(* CODESYS project DEMO.export

Project tree, tasks and I/O mapping:
  Device : Haitian E112C-0808N, Ningbo Anson CNC Technique CO., Ltd., version 1.1.32.0
      unmapped channels: DI, IN0_1_COUNT, IN2_3_COUNT, IN4_5_COUNT, IN6_7_COUNT, DO, OUT0_1_Pluse, OUT2_3_Pluse, OUT4_5_Pluse, OUT6_7_Pluse, IN, OUT
    application Application
      libraries: Standard, 3.5.18.0 (System); E112C Motion Control Lib, * (Haitian); E112C Communication  Lib, * (Haitian)
      task EtherCAT_Task (cyclic, interval 1000 µs, priority 1) calls DriverInHandlersEthercat, DriverOutHandlersEthercat, InitAxesProgram
      task MainTask (cyclic, interval 1 ms, priority 1) calls Motion_IO, Motion, Punch_PA, prTestFunction, DebugMode
      task Task1 (cyclic, interval 10 ms, priority 2) calls ModbusTCP_MasterPRG, prHMI, prCoolFan, prHMI_Error, SDO_test, prIOsetting_test, prModusTcp_Fanuc, SetPosition
      data type AxAbs
      data type Def_1
      data type Tcp_1
      BAK/
        program Punch_PA_1 [ST]
      FunctionBlock/
        function block FB_BLINK [ST]
        function block FB_CrankSliderHeight [ST]
        function block FB_HeightToAngle [ST]
        function block FB_Toggle [ST]
      MosbusTcp/
        program Modbus_Client_Fanuc [LD]: ACT_TRIG
        program prHMI [ST]
        program prHMI_Error [ST]
        program prModusTcp_Fanuc [ST]
      global variables AxisVars
      global variables GVL_Axis
      global variables GVL_HMI
      global variables GVL_PA
      global variables ModbusTCP_MasterVars
      program DebugMode [ST]: act_MoveNegative, act_MovePositive, act_SetHome
      program DriverInHandlersEthercat [ST]
      program DriverOutHandlersEthercat [ST]
      program InitAxesProgram [ST]
      program ModbusTCP_MasterPRG [ST]
      program Motion [ST]
      program Motion_IO [ST]
      program prCoolFan [ST]
      program prIOsetting_test [LD]: act_EtherCAT_monitor, act_Tcpdata
      program prTestFunction [ST]: act_Jump_To_PTE
      program Punch_PA [ST]: act_20_PunchA_GoPOP, act_21_PunchA_PunchA, act_22_PunchA_PunchB, act_31_PunchAB_PunchA, act_33_PunchAB_PunchB, act_41_PunchSoft_PunchA1, act_42_PunchSoft_PunchA2, act_43_PunchSoft_PunchA3, act_45_PunchSoft_PunchB1, act_46_PunchSoft_PunchB2, act_47_PunchSoft_PunchB3, act_7_GoPTE, act_Jump_To_PTE
      program SDO_test [LD]: act_Blink
      program SetHome [FBD]
      program SetPosition [?]
      program SetPosition0 [LD]
      program Test_Crank [ST]
      trace Trace (task MainTask): AxisVars.Axis0.AxisMotionState.ActPosition, ibPunch, qbReadyFeed, DriverOutHandlersEthercat.DriveOutHandler_Axis0.SetPosition
      global variables PersistentVars
    设备诊断
    设备组态
      EtherCAT机架
    轴配置
    资源使用表
    HT_LocalIO
        unmapped channels: DI, IN0_1_COUNT, IN2_3_COUNT, IN4_5_COUNT, IN6_7_COUNT, DO, OUT0_1_Pluse, OUT2_3_Pluse, OUT4_5_Pluse, OUT6_7_Pluse
    HT_LocalBus
        settings: EModuleCycle = 1000 us
      EM-DO16P [DO16 PNP] : EM-DO16P [DO16 PNP], Haitian, version 1.1.32.0
          unmapped channels: DO, DO
    HT_EtherCAT
      HT_Hi Drive v5.0 (TMS320F28377S, 16Bit Async, ET1100) : HT_Hi Drive v5.0 (TMS320F28377S, 16Bit Async, ET1100), HAITIAN DRIVE CO.,LTD, order no. Hi Drive v5.0, version Revision=16#00000001
          input  Application.DriverInHandlersEthercat.DriveInHandler_Axis0.StatusWord : UINT  // Status Word
          input  Application.DriverInHandlersEthercat.DriveInHandler_Axis0.ActPosition : DINT  // Position actual value
          input  Application.DriverInHandlersEthercat.DriveInHandler_Axis0.ActTorque : INT  // CI06 Current Iq actual value [A]
          input  Application.DriverInHandlersEthercat.DriveInHandler_Axis0.ActVelocity : DINT  // Velocity actual value [/10 r/min]
          input  Application.DriverInHandlersEthercat.DriveInHandler_Axis0.ModeOfDisplay : SINT  // Modes of operation display
          output Application.DriverOutHandlersEthercat.DriveOutHandler_Axis0.ControlWord : UINT  // Control Word
          output Application.DriverOutHandlersEthercat.DriveOutHandler_Axis0.SetTorque : INT  // Target torque [/10 %]
          output Application.DriverOutHandlersEthercat.DriveOutHandler_Axis0.SetPosition : DINT  // Target position
          output Application.DriverOutHandlersEthercat.DriveOutHandler_Axis0.SetVelocity : DINT  // Target velocity
          output Application.DriverOutHandlersEthercat.DriveOutHandler_Axis0.ModeOfOperation : SINT  // Modes of operation
          unmapped channels: RU09 Motor temperature [°C], Drive Error Code*, Max torque [/10 %], Elements
    HT_Ethernet
        settings: ip.ip = 192; ip.ip = 168; ip.ip = 1; ip.ip = 66; netmask.netmask = 255; netmask.netmask = 255; netmask.netmask = 255; netmask.netmask = 0; gateway.gateway = 192; gateway.gateway = 168; gateway.gateway = 1; gateway.gateway = 254; ModbusSlaveAddr = 0
    HT_EX1
    HT_EX2
    HT_Elink
        unmapped channels: IN, OUT
    HT_RS485_1
    HT_RS485_2
*)

// Device/Application/AxAbs
TYPE AxAbs :
STRUCT
	bExe :BOOL;
	Position :LREAL;
	Speed :LREAL;
	Acc :LREAL;
	Dcc :LREAL;
	Jerk :LREAL;
	Dir :MC_DIRECTION;
	BufferMode :MC_BUFFER_MODE;
	Done :BOOL;
	Busy :BOOL;
	Aborted :BOOL;
	Error :BOOL;
	ErrorID :WORD;
	Active :BOOL;
END_STRUCT
END_TYPE

// Device/Application/Def_1
TYPE Def_1 :
STRUCT
	
	Speed_Go_PTE :REAL :=100; //Go上死点PTE 速度
	Speed_Go_POP :REAL :=100; //上死点到预压POP 速度
 	
	
	Acc_Go_PTE : REAL :=3600;
	Acc_Go_POP : REAL :=3600;
	Acc_PunchA : REAL :=36000; //冲压A side
	Acc_PunchAB : REAL :=360000; //冲压AB side
	Acc_PunchSoft : REAL :=100000; //软冲 side
	
	CoolFan_Toff :INT :=10; //延时风扇关闭 sec 
	CoolFan_OnTemp :INT :=60; //自动打开温度
	
	PTE_Gap :REAL :=5; //到上死点0的到位窗口
	POP_Gap :REAL :=3; //到预压位角度的到位窗口 不是提前到位信号
	PUP_Gap :REAL :=2; //到下死点角度的到位窗口 不是提前到位信号	
	POP_ReadyWin_Punch :REAL :=10; //冲头冲压返回预压位置的提前到位窗口信号
	POP_ReadyWin_Mark :REAL :=5; //冲头冲压返回预压位置的提前到位窗口信号
	PunchSpeed_Max_Lim :REAL :=425; //冲头最高速度限制值
END_STRUCT
END_TYPE

// Device/Application/Tcp_1
TYPE Tcp_1 :
STRUCT
	bError :BOOL; 
	iRead_OK :INT; //读取数据正常计数器
	
	iPTE_mm :REAL :=32; //Data_1 换模位置 
	iPTE_deg :REAL; //Data_1 换模位置

	iPOP_mm :REAL;//Data_2 预压位置 上死点
	iPOP_deg :REAL;//Data_2 预压位置 上死点
	
	iPUP_mm :REAL; //Data_3 下压位置
	iPUP_deg :REAL;//Data_3 下压位置

	iReady_mm :REAL; //Data_4换模位置 ready 信号区域
	iReady_deg :REAL;//Data_4换模位置 ready 信号区域
	
	iDelayTime_ms : UINT;//Data_5  下压点延时

	iPunchSpeed_Trans :REAL; //Data_6 冲压速度	
	iPunchSpeed_Max :REAL; //Data_6 冲压速度
	iSoftPunch : INT;//Data_7 软冲模式
	
	iPSP1_mm :REAL ;//Data_8 软冲减速点1
	iPSP1_deg :REAL ;//Data_8 软冲减速点1
	
	iPunchSpeed :REAL; //Data_9 冲压穿板速度
	
	iFormMode :INT; //Data_10 压印模式 0-可调 1-机械点
	
	iPSP2_mm :REAL ;//Data_11 软冲减速点1
	iPSP2_deg :REAL ;//Data_11 软冲减速点1
	
	
	intermediate_iPOP_mm : WORD;
	intermediate_iReady_mm : WORD;
    intermediate_iPUP_mm : WORD;
    intermediate_iDelayTime_ms : WORD;
    intermediate_iPSP2_mm : WORD;
    intermediate_iPSP1_mm : WORD;
    intermediate_iPunchSpeed : WORD;
    intermediate_iPunchSpeed_Max : WORD;

END_STRUCT
END_TYPE

// Device/Application/AxisVars
//轴界面生成的轴全局变量
{attribute 'qualified_only'}
VAR_GLOBAL
	Axis0 : AXIS_REF := (AxisMotionState := (AxisNo := 0));
END_VAR

// Device/Application/GVL_Axis
VAR_GLOBAL
	MC_POWER0:MC_POWER;
	MC_RESET0: MC_Reset;
	MC_MODECONTROL0: MC_SetControllerMode;
	MC_STOP0: MC_Stop;
	MC_Abs_0: MC_MoveAbsolute;
	MC_Abs_1: MC_MoveAbsolute;
	MC_Abs_2: MC_MoveAbsolute;
	
	AxAbs_0 :AxAbs;
	AxAbs_1 :AxAbs;
	AxAbs_2 :AxAbs;
	
	POWER_ERROR:BOOL;
	rt_ibPunch:R_TRIG; //冲压信号
	rt_ibGoPOP:R_TRIG;//到预压位
	mGoPTE:BOOL;;//到换模位
	mGoPOP:BOOL;;//到预压位
	bPunchExe:BOOL;;//冲压信号
		
	Tcp :Tcp_1;
	Def :Def_1;
END_VAR

// Device/Application/GVL_HMI

VAR_GLOBAL
	bDebugModeEnable AT %MX3220.0:BOOL;;       // 打开调试功能按钮
    bDebugEnableBtn AT %MX3220.1: BOOL;       // 伺服使能按钮
    bHomeBtn AT %MX3220.2: BOOL;             // 驱动设零按钮
    bMovePosBtn AT %MX3220.3 : BOOL;       // 正向移动按钮
    bMoveNegBtn AT %MX3220.4: BOOL;       // 反向移动按钮 
	bSetPosBtn AT %MX3220.5: BOOL;       // 系统设零按钮
	rDebug_TargPos AT %MD806: REAL;
	
	bDebug_AFErr :BOOL;
	bDebug_MoveErr :BOOL;
	bDebug_SetHomeErr :BOOL;
	

END_VAR

// Device/Application/GVL_PA

VAR_GLOBAL
	//IX0 - 本地输入 
	ibModeSel_0 AT %IX0.0:BOOL; //工作模式信号—0
	ibModeSel_1 AT %IX0.1:BOOL; //工作模式信号—1
	ibModeSel_2 AT %IX0.2:BOOL; //工作模式信号—2
	ibPunch 	AT %IX0.3:BOOL ; //冲压信号
	ibGoPOP	 	AT %IX0.4:BOOL; //切换到上死点
	ibAF 		AT %IX0.5:BOOL ; //伺服使能
	ibSoftPun 	AT %IX0.6:BOOL; //软冲模式
	bMode_SetPos: BOOL;
	
	//QX0 - 本地输出 NPN模块	
	qPos_0 		AT %QX0.0:BOOL; //位置信号1—qx0
	qPos_1 		AT %QX0.1:BOOL; //位置信号2—qx0
	qReadyFeed 	AT %QX0.2:BOOL; //进料信号—qx0
	qError		AT %QX0.3 :BOOL; //冲头故障信号—qx0 
	qFan		AT %QX0.4 :BOOL; //风扇—qx0

	//QX20-21 - 扩展输出 PNP模块
	qbPos_0 	AT %QX20.0:BOOL; //位置信号1
	qbPos_1 	AT %QX20.1:BOOL; //位置信号2
	qbReadyFeed AT %QX20.2:BOOL; //进料信号
	qbError		AT %QX20.3 :BOOL; //冲头故障信号  
	qbFan		AT %QX20.4 :BOOL; //风扇
	
	qqbReadyFeed AT %QX20.5:BOOL; //进料信号
	
	iMotorTemp AT %IW15 :INT; //电机温度
	
	wModeSel :WORD;
	EXECUTE:BOOL:=TRUE;
	ibAtPTE:BOOL;
	ibAtPOP:BOOL;
	ibAtPUP:BOOL;
	byPos:BYTE;
	
	POP_Pos :REAL :=121;
	PUP_Pos :REAL :=180;
	PTE_Gap :REAL:=5; //In PTE position
	Punch_Speed :REAL :=400;//rpm
	PSP1_Pos :REAL;
	PSP2_Pos :REAL;
	PSP1_Speed:REAL :=100;
	PSP2_Speed:REAL :=350;
	
	ActPos :LREAL;//当前位置 角度
	PunHeight :LREAL;
	SetPosValue :LREAL;//设置当前位置值
	
	bReset :BOOL;
	bAFOn :BOOL;//使能轴
	wModeSel_Last :WORD;
	bMode_Switching :BOOL;
	bAF_Off :BOOL;//关使能
	bSetPosExe:BOOL;//执行重置绝对编码器位置
	bDriveError :BOOL;
	bDebugEnable : BOOL;
	
	bReady_OnFly :BOOL;//On Fast Read Check;
	bReady_Win :REAL :=10;//返回预压位置许可送料提前窗口
	
	iStep :INT :=0;
	bTest_OnOff AT %MX3200.0:BOOL;//测试模式开关
	bTest_AF AT %MX3200.1:BOOL;//测试模式使能
	bTest_iPOP AT %MX3200.2:BOOL;//测试模式 - 到预压点
	bTest  AT %MX3200.3:BOOL;//测试模式
	bTest_iPunch :BOOL; //测试模式-冲压信号
	bTest_GoPOP :BOOL; //测试模式 - 到预压点
	
	bIdle :BOOL;//通讯状态字
	bModbusSet_Error :BOOL;
	bModbusRead_Error :BOOL;
	bModbusWrite_Error :BOOL;
	
	Ecat_monitor :BYTE;//EtherCAT监控
	Ecat_Error :BOOL;//EtherCAT中断
	
END_VAR

// Device/Application/ModbusTCP_MasterVars
(* Auto-Generated Code by 'Modbus Configurator'.
 * DO NOT MODIFY HERE!
 * Changes will be overwritten.
 * If modification is required create a copy of this object. *)
VAR_GLOBAL
  Slave1TCPSetErrorId : WORD;
  Slave1Id1RBuff : ARRAY[0..9] OF WORD;
  Slave1Id1RErrorId : WORD;
  Slave1Id2WBuff : ARRAY[0..9] OF WORD;
  Slave1Id2WErrorId : WORD;
END_VAR

// Device/Application/PersistentVars
{attribute 'qualified_only'}
VAR_GLOBAL PERSISTENT RETAIN
	socket:byte;
END_VAR

// Device/Application/DriverInHandlersEthercat
(* Auto-Generated Code by 'Axes Configurator'.
 * DO NOT MODIFY HERE!
 * Changes will be overwritten.
 * If modification is required create a copy of this object. *)
PROGRAM DriverInHandlersEthercat
VAR
	DriveInHandler_Axis0: MC_AxisDataIn;
END_VAR

(* Auto-Generated Code by 'Axes Configurator'.
 * DO NOT MODIFY HERE!
 * Changes will be overwritten.
 * If modification is required create a copy of this object. *)

DriveInHandler_Axis0(
	Axis:= AxisVars.Axis0,
	Enable:= 1, 
	ControlPeriod:= 1000,
	VirtualEnable:= False,
	ServoVelUnit:= 1, 
	StatusWord:=, 
	ActPosition:=, 
	ActVelocity:=, 
	ActTorque:=, 
	ModeOfDisplay:=, 
	FollowingError:=, 
	TouchProbeStatus:=, 
	TouchProbe1RisingEdge:=, 
	TouchProbe1FallingEdge:=, 
	TouchProbe2RisingEdge:=, 
	TouchProbe2FallingEdge:=, 
	Done => , 
	Error => , 
	ErrorID => 
);

END_PROGRAM

// Device/Application/DriverOutHandlersEthercat
(* Auto-Generated Code by 'Axes Configurator'.
 * DO NOT MODIFY HERE!
 * Changes will be overwritten.
 * If modification is required create a copy of this object. *)
PROGRAM DriverOutHandlersEthercat
VAR
	DriveOutHandler_Axis0: MC_AxisDataOut;
END_VAR

(* Auto-Generated Code by 'Axes Configurator'.
 * DO NOT MODIFY HERE!
 * Changes will be overwritten.
 * If modification is required create a copy of this object. *)

DriveOutHandler_Axis0(
	Axis:= AxisVars.Axis0,
	Enable:= 1, 
	Done => , 
	Error => , 
	ErrorID => , 
	ControlWord =>, 
	SetPosition =>, 
	SetVelocity =>, 
	SetTorque =>, 
	ModeOfOperation =>, 
	TouchProbeFun =>, 
	AddVelValue =>, 
	AddTorqueValue =>, 
	Var1 => , 
	Var2 => 
);

END_PROGRAM

// Device/Application/SetPosition
PROGRAM SetPosition
VAR
	
	bKey_SetPos: BOOL;
	rValue_SetPos: REAL :=0;
	
	MC_Home0: MC_Home;
	
END_VAR

(* body of a kind this reader does not render *)

END_PROGRAM

// Device/Application/InitAxesProgram
(* Auto-Generated Code by 'Axes Configurator'.
 * DO NOT MODIFY HERE!
 * Changes will be overwritten.
 * If modification is required create a copy of this object. *)
PROGRAM InitAxesProgram
VAR_OUTPUT
	Done: BOOL;
	Error: BOOL;
END_VAR
VAR
	InitAxis0Axis: MC_AxisParaInit;
	InitAxis0Cmd: BOOL := TRUE;
END_VAR

(* Auto-Generated Code by 'Axes Configurator'.
 * DO NOT MODIFY HERE!
 * Changes will be overwritten.
 * If modification is required create a copy of this object. *)
InitAxis0Axis(
	Axis:= AxisVars.Axis0,
	Execute:= InitAxis0Cmd, 
	ActiveFlag:= 1, 
	MotionType:= 1, 
	VelocityType:= 0, 
	ControllerMode:= 0, 
	EncoderType:= 1, 
	IgnoreSofwareLimit:= , 
	InputScale:= 8388608, 
	OutputScale:= 8388608, 
	GearScale:= 360, 
	BackLash:= , 
	ModuloValue:= 360, 
	MaxPos:= , 
	MinPos:= , 
	MaxVel:= 3600, 
	MaxAcc:= 36000000, 
	MaxDec:= 36000000, 
	MaxJerk:= 36000000, 
	MinError:= 100000, 
	MaxError:= 100000, 
	MotorOffset:= , 
	Done => , 
	Error => , 
	ErrorID => 
);

IF(InitAxis0Axis.Done) THEN
	Done := TRUE;
END_IF

IF(InitAxis0Axis.Error) THEN
	Error := TRUE;
END_IF

END_PROGRAM

// Device/Application/Motion_IO
//Motion 高速IO及计算
PROGRAM Motion_IO
VAR
	mReady :BOOL;
	
END_VAR

//当前位置
ActPos :=AxisVars.Axis0.AxisMotionState.ActPosition;

//冲压及预压信号触发
rt_ibPunch(CLK:= (ibPunch OR bTest_iPunch) AND mGoPOP AND FALSE, Q=> );
IF (ibPunch OR bTest_iPunch) AND mGoPOP THEN 
	bPunchExe:=TRUE;
ELSE
	bPunchExe :=FALSE;	
END_IF
IF mGoPTE THEN 
	bPunchExe :=FALSE;
END_IF

//rt_ibGoPOP(CLK:= ibGoPOP OR bTest_iPOP, Q=> );
IF ibGoPOP OR bTest_GoPOP THEN 
	mGoPOP:=TRUE;
	mGoPTE:=FALSE;	
ELSE
	mGoPOP:=FALSE;
	mGoPTE:=TRUE;
END_IF

//Check at PTE 是否在上死点位置
IF ABS(ActPos - 0)<Def.PTE_Gap THEN
	ibAtPTE:=TRUE;
ELSE
	IF ABS(ActPos - 360)<Def.PTE_Gap THEN
		ibAtPTE:=TRUE;
	ELSE
		ibAtPTE:=FALSE;	
	END_IF
END_IF

//Check at 是否发出送料信号
IF ActPos <(Tcp.iPOP_deg + Def.POP_Gap) OR (ActPos>180 
		AND ActPos>(360-Tcp.iPOP_deg - Def.POP_Gap)) OR ibAtPTE THEN
	mReady:=TRUE;
ELSE
	IF bReady_OnFly AND 
	((ActPos <(Tcp.iPOP_deg+bReady_Win)) OR (ActPos>180 AND ActPos>(360-Tcp.iPOP_deg-bReady_Win) ))  THEN
		mReady:=TRUE;
	ELSE
		mReady:=FALSE;	
	END_IF
END_IF
qbReadyFeed :=mReady;
qqbReadyFeed :=mReady;

//Check at POP 是否在预压点位置
ibAtPOP :=mReady AND NOT ibAtPTE;

//Check at PUP 是否在下死点位置
IF (ActPos >(Tcp.iPUP_deg - Def.PUP_Gap)) AND (ActPos <(Tcp.iPUP_deg + Def.PUP_Gap)) THEN
	ibAtPUP:=TRUE;
ELSE
	ibAtPUP:=FALSE;
END_IF

//输出映射到 本地QX0-NPN模块
CASE byPos OF
	1:
		qPos_0 :=TRUE;
		qPos_1 :=FALSE;
	2:
		qPos_0 :=FALSE;
		qPos_1 :=TRUE;
	4:
		qPos_0 :=TRUE;
		qPos_1 :=TRUE;		
ELSE
		qPos_0 :=FALSE;
		qPos_1 :=FALSE;
END_CASE;

//输出映射到 LocalBus QX20/21-PNP模块
qbPos_0 :=qPos_0;
qbPos_1 :=qPos_1;


//输出映射到 本地QX0-NPN模块
qReadyFeed :=qbReadyFeed;
qError :=qbError;
qFan :=qbFan;

END_PROGRAM

// Device/Application/Motion
// PLCOpen 功能块
PROGRAM Motion
VAR
	POWER_ENABLE0:BOOL;
	POWER_STATUS0:BOOL;
	POWER_ERRORID:WORD;
	
	RESET_EXECUTE0:BOOL;
	RESET_DONE0:BOOL;
	RESET_BUSY0:BOOL;
	RESET_ERROR0:BOOL;
	RESET_ERRORID0:WORD;
	
	STOP_EXECUTE0:BOOL;
	STOP_DECELERATION0:LREAL:=10;
	STOP_JERK0:LREAL:=10;
	STOP_DONE0:BOOL;
	STOP_BUSY0:BOOL;
	STOP_COMMANDABORTED:BOOL;
	STOP_ERROR0:BOOL;
	STOP_ERRORID0:WORD;
	
	MODE_EXECUTE0:BOOL;
	MODE_CONTROLLERMODE:MC_CONTROLLER_MODE;
	MODE_DONE0:BOOL;
	MODE_BUSY0:BOOL;
	MODE_ERROR0:BOOL;
	MODE_ERRORID0:WORD;
	
	ABSOLUTE_EXECUTE0:BOOL;
	ABSOLUTE_POSITION0:LREAL:=90;
	ABSOLUTE_VELOCITY0:LREAL:=1800;
	ABSOLUTE_ACCELERATION0:LREAL:=36000000;
	ABSOLUTE_DECELERATION0:LREAL:=36000000;
	ABSOLUTE_JERK0:LREAL:=360000000;
	ABSOLUTE_DIRECTION0:MC_DIRECTION;
	ABSOLUTE_BUFFERMODE0:MC_BUFFER_MODE;
	ABSOLUTE_DONE0:BOOL;
	ABSOLUTE_BUSY0:BOOL;
	ABSOLUTE_ACTIVE0:BOOL;
	ABSOLUTE_COMMANDABORTED0:BOOL;
	ABSOLUTE_ERROR0:BOOL;
	ABSOLUTE_ERRORID0:WORD;
	
	ABSOLUTE_EXECUTE1:BOOL;
	ABSOLUTE_POSITION1:LREAL:=180;
	ABSOLUTE_VELOCITY1:LREAL:=360;
	ABSOLUTE_ACCELERATION1:LREAL:=36000000;
	ABSOLUTE_DECELERATION1:LREAL:=36000000;
	ABSOLUTE_JERK1:LREAL:=360000000;
	ABSOLUTE_DIRECTION1:MC_DIRECTION;
	ABSOLUTE_BUFFERMODE1:MC_BUFFER_MODE;
	ABSOLUTE_DONE1:BOOL;
	ABSOLUTE_BUSY1:BOOL;
	ABSOLUTE_ACTIVE1:BOOL;
	ABSOLUTE_COMMANDABORTED1:BOOL;
	ABSOLUTE_ERROR1:BOOL;
	ABSOLUTE_ERRORID1:WORD;
	
	ABSOLUTE_EXECUTE2:BOOL;
	ABSOLUTE_POSITION2:LREAL:=360;
	ABSOLUTE_VELOCITY2:LREAL:=2880;
	ABSOLUTE_ACCELERATION2:LREAL:=36000000;
	ABSOLUTE_DECELERATION2:LREAL:=36000000;
	ABSOLUTE_JERK2:LREAL:=360000000;
	ABSOLUTE_DIRECTION2:MC_DIRECTION;
	ABSOLUTE_BUFFERMODE2:MC_BUFFER_MODE;
	ABSOLUTE_DONE2:BOOL;
	ABSOLUTE_BUSY2:BOOL;
	ABSOLUTE_ACTIVE2:BOOL;
	ABSOLUTE_COMMANDABORTED2:BOOL;
	ABSOLUTE_ERROR2:BOOL;
	ABSOLUTE_ERRORID2:WORD;
	

	a AT %MD0:DWORD;
	//a1 AT MW1 :WORD;;
	a2 AT %MW2:DWORD;
	a3 AT %MW4:DWORD;

	icounter:int;

END_VAR


MC_POWER0(
	Axis:= AxisVars.Axis0, 	
	Enable:= (bAFOn AND NOT POWER_ERROR AND NOT bAF_Off) OR bDebugEnable, 
	Status=> POWER_STATUS0, 	Valid=> ,	
	Error=> POWER_ERROR,	ErrorID=> POWER_ERRORID);
	
MC_RESET0(
	Axis:= AxisVars.Axis0, 
	Execute:= RESET_EXECUTE0 OR bReset , 
	Done=> RESET_DONE0, 	Busy=> RESET_BUSY0,	
	Error=> RESET_ERROR0,	ErrorID=> RESET_ERRORID0);
	
MC_STOP0(
	Axis:= AxisVars.Axis0, 	Execute:= STOP_EXECUTE0, 
	Deceleration:= STOP_DECELERATION0, 
	Jerk:= STOP_JERK0, 
	Done=> STOP_DONE0, 	Busy=> STOP_BUSY0,	
	CommandAborted=> STOP_COMMANDABORTED,	
	Error=> STOP_ERROR0, 
	ErrorID=> STOP_ERRORID0);
	
MC_MODECONTROL0(
	Axis:= AxisVars.Axis0, 	Execute:= MODE_EXECUTE0, 	
	ControllerMode:= MODE_CONTROLLERMODE, 
	Done=> MODE_DONE0, 	Busy=> MODE_BUSY0,	
	Error=> MODE_ERROR0,	ErrorID=> MODE_ERRORID0);

MC_Abs_0(
	Axis:= AxisVars.Axis0, 
	Execute:= AxAbs_0.bExe, 	Position:= AxAbs_0.Position, 
	Velocity:= AxAbs_0.Speed, 	
	Acceleration:= AxAbs_0.Acc, 	Deceleration:= AxAbs_0.Dcc, 
	Jerk:= AxAbs_0.Jerk, 	Direction:= AxAbs_0.Dir,	
	BufferMode:= AxAbs_0.BufferMode, 
	Done=> AxAbs_0.Done, 	Busy=> AxAbs_0.Busy,	Active=> AxAbs_0.Active,
	CommandAborted=> AxAbs_0.Aborted,	
	Error=> AxAbs_0.Error,	ErrorID=> AxAbs_0.ErrorID);
	
MC_Abs_1(
	Axis:= AxisVars.Axis0, 
	Execute:= AxAbs_1.bExe, 	Position:= AxAbs_1.Position, 
	Velocity:= AxAbs_1.Speed, 	
	Acceleration:= AxAbs_1.Acc, 	Deceleration:= AxAbs_1.Dcc, 
	Jerk:= AxAbs_1.Jerk, 	Direction:= AxAbs_1.Dir,	
	BufferMode:= AxAbs_1.BufferMode, 
	Done=> AxAbs_1.Done, 	Busy=> AxAbs_1.Busy,	Active=> AxAbs_1.Active,
	CommandAborted=> AxAbs_1.Aborted,	
	Error=> AxAbs_1.Error,	ErrorID=> AxAbs_1.ErrorID);
	
MC_Abs_2(
	Axis:= AxisVars.Axis0, 
	Execute:= AxAbs_2.bExe, 	Position:= AxAbs_2.Position, 
	Velocity:= AxAbs_2.Speed, 	
	Acceleration:= AxAbs_2.Acc, 	Deceleration:= AxAbs_2.Dcc, 
	Jerk:= AxAbs_2.Jerk, 	Direction:= AxAbs_2.Dir,	
	BufferMode:= AxAbs_2.BufferMode, 
	Done=> AxAbs_2.Done, 	Busy=> AxAbs_2.Busy,	Active=> AxAbs_2.Active,
	CommandAborted=> AxAbs_2.Aborted,	
	Error=> AxAbs_2.Error,	ErrorID=> AxAbs_2.ErrorID);

END_PROGRAM

// Device/Application/Punch_PA
PROGRAM Punch_PA
VAR
	iCounter :UINT :=0;
	iDelayTime_ms : UINT :=0;
	actModeSet :INT;
	bFreeMark :bool; //自由打标模式激活中
END_VAR

IF NOT bAFOn  THEN
	iStep := iCounter:=0;
END_IF 

CASE iStep OF
	0://Power Off, reset data
		AxAbs_0.bExe := AxAbs_1.bExe :=AxAbs_2.bExe := bAF_Off := bReset :=FALSE;
		IF bAFOn AND MC_POWER0.Error THEN
			iCounter :=0;
			iStep :=1;
		END_IF
		IF bAFOn AND NOT MC_POWER0.Error AND AxisVars.Axis0.AxisMotionState.ServoEnabled AND NOT bMode_SetPos THEN
			iStep :=7;
		END_IF
	1:
		bReset := bAF_Off :=TRUE;
		iCounter :=iCounter +1;
		IF iCounter >1000 AND MC_RESET0.Done THEN
			bReset :=FALSE;
			iStep :=2; iCounter :=0;
		END_IF
	2: bReset :=FALSE; bAF_Off :=TRUE;
		iCounter :=iCounter +1;
		IF iCounter >1000 THEN
			bAF_Off :=FALSE;
			iStep :=0; iCounter :=0;//返回0步
		END_IF
		
	7://PrePTE
		act_7_GoPTE();
		AxAbs_0.bExe := AxAbs_1.bExe :=AxAbs_2.bExe :=FALSE;
		iCounter:= iCounter +1;
		IF iCounter>100 THEN
			iStep :=10;
			iCounter :=0;
		END_IF	
		
	10://Back to PTE
		IF mGoPTE THEN
			AxAbs_0.bExe :=TRUE;		
		END_IF
		IF MC_Abs_0.Active THEN
			AxAbs_0.bExe :=FALSE;
		END_IF
		IF MC_Abs_0.Done AND  ibAtPTE THEN
			AxAbs_0.bExe :=FALSE;
			iCounter :=iCounter+1;
			IF iCounter>50 THEN
				iStep :=15;
				iCounter :=0;			
			END_IF
		END_IF
	
	15://Waiting for Switching Mode
		bReady_OnFly :=FALSE;
		CASE wModeSel OF
				0://Punch-A Side	Forming/Wheel/Scribe
					IF mGoPOP THEN
						iDelayTime_ms :=Tcp.iDelayTime_ms;
						actModeSet :=0;
						bReady_Win:=0;//提前到位=0
						iStep :=20;
					END_IF
			
				1://Undefinition
			
				2://Free mark
					IF mGoPOP THEN
						iDelayTime_ms :=0;
						actModeSet :=2;//标记 自由打标
						bReady_Win:=Def.POP_ReadyWin_Mark;//使用打标提前到位窗
						bFreeMark :=TRUE; //设置自由打标控制参数
						iStep :=50;
					END_IF
				
				3://Punch-AB Side
					IF mGoPOP THEN
						actModeSet :=3;
						IF ibSoftPun THEN
							bReady_Win:=0;//软冲冲压提前到位窗=0
							iStep :=40;
						ELSE
//							bReady_Win:=Def.POP_ReadyWin_Punch;//冲压使用默认冲压提前到位窗
							bReady_Win:=Tcp.iReady_deg;//冲压使用上位传输冲压提前到位窗
							iStep :=30;
						END_IF
					END_IF
					
				4://Round 
				
				5://Mark-With POP
					IF mGoPOP THEN
						iDelayTime_ms :=0;
						actModeSet :=5;//标记 打标模式
						bReady_Win:=Def.POP_ReadyWin_Mark;//使用打标提前到位窗
						iStep :=20;
					END_IF

		END_CASE
		
	20://Punch - Aside - step0 - 到预压POP
		act_20_PunchA_GoPOP();
		IF mGoPOP THEN 
			AxAbs_0.bExe :=TRUE;
		END_IF
		IF MC_Abs_0.Active THEN
			AxAbs_0.bExe :=FALSE;
		END_IF	
		act_Jump_To_PTE();
		IF MC_Abs_0.Done THEN
			AxAbs_0.bExe :=FALSE;
			iCounter :=iCounter+1;
			IF iCounter>100 THEN
				iStep :=21;	iCounter :=0;
			END_IF
		END_IF		
		
	21://Punch - Aside - step1 - 等待冲压信号 Pun-ibPunch 
		act_21_PunchA_PunchA();
		AxAbs_0.bExe :=FALSE;	
		act_Jump_To_PTE();
		IF rt_ibPunch.Q OR bPunchExe THEN
			bPunchExe :=FALSE;				
			bReady_OnFly :=FALSE;
			iCounter:=0; iStep :=22;
		END_IF
		
	22://Punch - Aside - step2
		act_22_PunchA_PunchB();
		AxAbs_0.bExe :=TRUE;
		IF MC_Abs_0.Active THEN
			AxAbs_0.bExe :=FALSE;
		END_IF	
		AxAbs_1.bExe :=FALSE;
		act_Jump_To_PTE();
		IF MC_Abs_0.Done THEN
			AxAbs_0.bExe :=FALSE;
			iCounter := iCounter + 1;
			IF iCounter >= iDelayTime_ms/3 THEN
				iCounter:=0; iStep :=23;			
			END_IF
		END_IF
		
	23://Punch - Aside - step3	
		bReady_OnFly :=TRUE;
		act_Jump_To_PTE();
		AxAbs_1.bExe :=TRUE;
		IF MC_Abs_1.Active THEN
			AxAbs_1.bExe :=FALSE;
		END_IF		
		IF MC_Abs_1.Done THEN
			AxAbs_1.bExe :=FALSE;
			iStep :=21;			
		END_IF		
	
	
	30://Punch - ABside - step0 - Go POP
		act_20_PunchA_GoPOP();
		act_Jump_To_PTE();
		IF mGoPOP THEN 
			AxAbs_0.bExe :=TRUE;
		END_IF 
		IF MC_Abs_0.Active THEN
			AxAbs_0.bExe :=FALSE;
		END_IF	
		IF MC_Abs_0.Done THEN
			AxAbs_0.bExe :=FALSE;
			iCounter :=iCounter+1;
			IF iCounter>100 THEN
				iStep :=31;	iCounter :=0;			
			END_IF
		END_IF	
		
	31://Punch - ABside - step1 - Wating Pun-ibPunch
		act_31_PunchAB_PunchA();
		AxAbs_0.bExe :=FALSE;	
		act_Jump_To_PTE();
		IF rt_ibPunch.Q OR bPunchExe THEN
			bPunchExe :=FALSE;
			bReady_OnFly :=FALSE;
			iStep :=32;
		END_IF
		
	32://Punch - ABside - step1 - Wating Pun-ibPunch
		AxAbs_0.bExe :=TRUE;	
		IF	ActPos>180 THEN
			bReady_OnFly :=TRUE;
		END_IF
		act_Jump_To_PTE();
		IF MC_Abs_0.Active THEN
			AxAbs_0.bExe :=FALSE;
		END_IF	
		IF MC_Abs_0.Done THEN
			AxAbs_0.bExe :=FALSE;
			iStep :=33;	iCounter :=0;			
		END_IF		
		
	33://Punch - ABside - step1 - Wating Pun-ibPunch
		act_33_PunchAB_PunchB();
		AxAbs_0.bExe :=FALSE;	
		act_Jump_To_PTE();
		IF rt_ibPunch.Q OR bPunchExe THEN
			bPunchExe :=FALSE;
			bReady_OnFly :=FALSE;
			iStep :=34;
		END_IF
		
	34://Punch - ABside - step1 - Wating Pun-ibPunch
		AxAbs_0.bExe :=TRUE;
		IF	ActPos<180 THEN
			bReady_OnFly :=TRUE;
		END_IF	
		act_Jump_To_PTE();
		IF MC_Abs_0.Active THEN
			AxAbs_0.bExe :=FALSE;
		END_IF	
		IF MC_Abs_0.Done THEN
			AxAbs_0.bExe :=FALSE;
			iStep :=31;	iCounter :=0;			
		END_IF	



	40://Punch - ABside SoftPunch - step0 - Go POP
		act_20_PunchA_GoPOP();
		act_Jump_To_PTE();
		IF mGoPOP THEN 
			AxAbs_0.bExe :=TRUE;
		END_IF 	
		IF MC_Abs_0.Active THEN
			AxAbs_0.bExe :=FALSE;
		END_IF	
		IF MC_Abs_0.Done THEN
			AxAbs_0.bExe :=FALSE;
			iCounter :=iCounter+1;
			IF iCounter>100 THEN
				iStep :=41;	iCounter :=0;			
			END_IF
		END_IF	
		
		
		
	41:
		act_41_PunchSoft_PunchA1();
		AxAbs_0.bExe :=FALSE;	
		act_Jump_To_PTE();
		IF rt_ibPunch.Q OR bPunchExe THEN
			bPunchExe :=FALSE;
			bReady_OnFly :=FALSE;
			iStep :=42;
		END_IF
		
		
		
	42:
		act_42_PunchSoft_PunchA2();
		act_Jump_To_PTE();
		AxAbs_0.bExe :=TRUE;
		AxAbs_1.bExe :=FALSE;
		IF MC_Abs_0.Active THEN
			AxAbs_0.bExe :=FALSE;
		END_IF	
		IF MC_Abs_0.Done THEN
			AxAbs_0.bExe :=FALSE;
			iStep :=43;	iCounter :=0;			
		END_IF	
		
		
		
	43:
		act_43_PunchSoft_PunchA3();
		act_Jump_To_PTE();
		AxAbs_1.bExe :=TRUE;
		AxAbs_2.bExe :=FALSE;
		IF MC_Abs_1.Active THEN
			AxAbs_1.bExe :=FALSE;
		END_IF	
		IF MC_Abs_1.Done THEN
			AxAbs_1.bExe :=FALSE;
			iStep :=44;	iCounter :=0;			
		END_IF
		
		
		
	44:
		AxAbs_2.bExe :=TRUE;
		IF	ActPos>180 THEN
			bReady_OnFly :=TRUE;
		END_IF		
		act_Jump_To_PTE();
		IF MC_Abs_2.Active THEN
			AxAbs_2.bExe :=FALSE;
		END_IF	
		IF MC_Abs_2.Done THEN
			AxAbs_2.bExe :=FALSE;
			iStep :=45;	iCounter :=0;			
		END_IF
		
		
		
	45:
		act_45_PunchSoft_PunchB1();
		AxAbs_0.bExe :=FALSE;
		act_Jump_To_PTE();	
		IF rt_ibPunch.Q OR bPunchExe THEN
			bPunchExe :=FALSE;
			bReady_OnFly :=FALSE;
			iStep :=46;
		END_IF
	


	46:
		act_46_PunchSoft_PunchB2();
		act_Jump_To_PTE();
		AxAbs_0.bExe :=TRUE;
		AxAbs_1.bExe :=FALSE;
		IF MC_Abs_0.Active THEN
			AxAbs_0.bExe :=FALSE;
		END_IF	
		IF MC_Abs_0.Done THEN
			AxAbs_0.bExe :=FALSE;
			iStep :=47;	iCounter :=0;			
		END_IF	
		
		
		
	47:
		act_47_PunchSoft_PunchB3();
		act_Jump_To_PTE();
		AxAbs_1.bExe :=TRUE;
		AxAbs_2.bExe :=FALSE;
		IF MC_Abs_1.Active THEN
			AxAbs_1.bExe :=FALSE;
		END_IF	
		IF MC_Abs_1.Done THEN
			AxAbs_1.bExe :=FALSE;
			iStep :=48;	iCounter :=0;			
		END_IF
		
		
		
	48:
		AxAbs_2.bExe :=TRUE;
		IF	ActPos<180 THEN
			bReady_OnFly :=TRUE;
		END_IF		
		act_Jump_To_PTE();
		IF MC_Abs_2.Active THEN
			AxAbs_2.bExe :=FALSE;
		END_IF	
		IF MC_Abs_2.Done THEN
			AxAbs_2.bExe :=FALSE;
			iStep :=41;	iCounter :=0;			
		END_IF


	50://Free Mark - step0 - Go POP
		act_20_PunchA_GoPOP();
		IF mGoPOP THEN 
			AxAbs_0.bExe :=TRUE;
		END_IF
		IF MC_Abs_0.Active THEN
			AxAbs_0.bExe :=FALSE;
		END_IF	
		act_Jump_To_PTE();
		IF MC_Abs_0.Done THEN
			AxAbs_0.bExe :=FALSE;
			iCounter :=iCounter+1;
			IF iCounter>100 THEN
				iStep :=51;	iCounter :=0;
			END_IF
		END_IF		

	51://Free Mark - Aside - step1 - 等待冲压信号 Pun-ibPunch 
		act_21_PunchA_PunchA();
		AxAbs_0.bExe :=FALSE;	
		act_Jump_To_PTE();
		iCounter :=iCounter +1;
		IF rt_ibPunch.Q OR bPunchExe THEN
			bReady_OnFly :=FALSE;
			iCounter:=0; iStep :=52;
		END_IF

	52://Free Mark - Aside - step2
		act_22_PunchA_PunchB();
		AxAbs_0.bExe :=TRUE;
		IF MC_Abs_0.Active THEN
			AxAbs_0.bExe :=FALSE;
		END_IF	
		AxAbs_1.bExe :=FALSE;
		act_Jump_To_PTE();
		IF MC_Abs_0.Done THEN
			AxAbs_0.bExe :=FALSE;
			iStep :=53;			
		END_IF

	53://Free Mark - Aside - step3	
		bReady_OnFly :=TRUE;
		act_Jump_To_PTE();
		AxAbs_1.bExe :=TRUE;
		IF MC_Abs_1.Active THEN
			AxAbs_1.bExe :=FALSE;
		END_IF		
		IF MC_Abs_1.Done THEN
			AxAbs_1.bExe :=FALSE;
			iStep :=51;			
		END_IF	
	
	(*
	20://PreStep for Switching Mode
		AxAbs_0.Position :=80;		AxAbs_0.Speed :=100;
		AxAbs_0.Acc := AxAbs_0.Dcc :=360000; AxAbs_0.Jerk :=3600000;
		AxAbs_0.BufferMode :=MC_BUFFER_MODE.Buffered;
		AxAbs_0.Dir := MC_DIRECTION.mcPositive;	

		AxAbs_0.bExe :=TRUE;
		IF MC_Abs_0.Active THEN
			AxAbs_0.bExe :=FALSE;
		END_IF	
		IF MC_Abs_0.Done THEN
			iStep :=21;
		END_IF	
		
		
	21:
		AxAbs_1.Position :=180;		AxAbs_1.Speed :=20;
		AxAbs_1.Acc := AxAbs_1.Dcc :=360000; AxAbs_1.Jerk :=3600000;
		AxAbs_1.BufferMode :=MC_BUFFER_MODE.Aborting;
		AxAbs_1.Dir := MC_DIRECTION.mcPositive;	
		AxAbs_1.bExe :=TRUE;
		IF MC_Abs_1.Active THEN
			AxAbs_1.bExe :=FALSE;
		END_IF
		IF MC_Abs_1.Done THEN
			iStep :=25;
			AxAbs_1.bExe :=FALSE;
		END_IF
	25:
		iCounter :=iCounter+1;
		IF iCounter>500 THEN
			iStep :=30;
			iCounter :=0;
		END_IF
		
	30://PreStep for Switching Mode
		AxAbs_0.Position :=0;		AxAbs_0.Speed :=100;
		AxAbs_0.Acc := AxAbs_0.Dcc :=360000; AxAbs_0.Jerk :=3600000;
		AxAbs_0.BufferMode :=MC_BUFFER_MODE.Aborting;
		AxAbs_0.Dir := MC_DIRECTION.mcNegative;
		AxAbs_0.bExe :=FALSE;AxAbs_1.bExe :=FALSE;

		iCounter :=iCounter+1;
		IF iCounter>500 THEN
			iStep :=31;
			iCounter :=0;
		END_IF
		
	31:	
		AxAbs_0.bExe :=TRUE;
		IF MC_Abs_0.Active THEN
			AxAbs_0.bExe :=FALSE;
		END_IF		
		IF MC_Abs_0.Done THEN
			iStep :=35;
			AxAbs_0.bExe :=FALSE;		
		END_IF
	35:
		iCounter :=iCounter+1;
		AxAbs_0.BufferMode :=MC_BUFFER_MODE.Buffered;
		AxAbs_1.BufferMode :=MC_BUFFER_MODE.Aborting;
		AxAbs_0.bExe :=FALSE;
		AxAbs_1.bExe :=FALSE;
		IF iCounter>1000 THEN
			iStep :=20;
			iCounter :=0;
		END_IF		
		*)
		
END_CASE

ACTION act_20_PunchA_GoPOP:
// 20 - Punch A side Go POP 预压位置

AxAbs_0.Position :=Tcp.iPOP_deg;		
AxAbs_0.Speed :=Def.Speed_Go_POP*6;
AxAbs_0.Acc := AxAbs_0.Dcc :=Def.Acc_Go_POP; 
AxAbs_0.Jerk :=3600000;
AxAbs_0.BufferMode :=MC_BUFFER_MODE.Aborting;
AxAbs_0.Dir := MC_DIRECTION.mcPositive;
END_ACTION

ACTION act_21_PunchA_PunchA:
// 21 - Punch A Side Watiing bPunching 到下死点 PUP
AxAbs_0.Position :=Tcp.iPUP_deg;		
AxAbs_0.Speed :=Tcp.iPunchSpeed_Max*6;
AxAbs_0.Acc := AxAbs_0.Dcc := Def.Acc_PunchA; 
AxAbs_0.Jerk :=3600000;
AxAbs_0.BufferMode :=MC_BUFFER_MODE.Aborting;
AxAbs_0.Dir := MC_DIRECTION.mcPositive;
END_ACTION

ACTION act_22_PunchA_PunchB:
// 22 _ Punch A Side , Punch Step 2
AxAbs_1.Position :=Tcp.iPOP_deg;		
AxAbs_1.Speed :=Tcp.iPunchSpeed_Max*6;
AxAbs_1.Acc := AxAbs_1.Dcc :=Def.Acc_PunchA; 
AxAbs_1.Jerk :=3600000;
AxAbs_1.BufferMode :=MC_BUFFER_MODE.Aborting;
AxAbs_1.Dir := MC_DIRECTION.mcNegative;
END_ACTION

ACTION act_31_PunchAB_PunchA:
AxAbs_0.Position :=360 - TCP.iPOP_deg;		
AxAbs_0.Speed :=TCP.iPunchSpeed_Max*6;
AxAbs_0.Acc := AxAbs_0.Dcc :=Def.Acc_PunchAB; 
AxAbs_0.Jerk :=3600000;
AxAbs_0.BufferMode :=MC_BUFFER_MODE.Aborting;
AxAbs_0.Dir := MC_DIRECTION.mcPositive;
END_ACTION

ACTION act_33_PunchAB_PunchB:
AxAbs_0.Position :=TCP.iPOP_deg;		
AxAbs_0.Speed :=TCP.iPunchSpeed_Max*6;
AxAbs_0.Acc := AxAbs_0.Dcc :=Def.Acc_PunchAB; 
AxAbs_0.Jerk :=3600000;
AxAbs_0.BufferMode :=MC_BUFFER_MODE.Aborting;
AxAbs_0.Dir := MC_DIRECTION.mcNegative;
END_ACTION

ACTION act_41_PunchSoft_PunchA1:
AxAbs_0.Position :=TCP.iPSP1_deg;		
AxAbs_0.Speed :=TCP.iPunchSpeed_Max*6;
AxAbs_0.Acc := AxAbs_0.Dcc :=Def.Acc_PunchSoft; 
AxAbs_0.Jerk :=3600000;
AxAbs_0.BufferMode :=MC_BUFFER_MODE.BlendingLow;
AxAbs_0.Dir := MC_DIRECTION.mcPositive;
END_ACTION

ACTION act_42_PunchSoft_PunchA2:
AxAbs_1.Position :=TCP.iPSP2_deg;		
AxAbs_1.Speed :=TCP.iPunchSpeed*6;
AxAbs_1.Acc := AxAbs_1.Dcc :=Def.Acc_PunchSoft; 
AxAbs_1.Jerk :=3600000;
AxAbs_1.BufferMode :=MC_BUFFER_MODE.BlendingLow;
AxAbs_1.Dir := MC_DIRECTION.mcPositive;
END_ACTION

ACTION act_43_PunchSoft_PunchA3:
AxAbs_2.Position :=360 - TCP.iPOP_deg;		
AxAbs_2.Speed :=TCP.iPunchSpeed_Max*6;
AxAbs_2.Acc := AxAbs_2.Dcc :=Def.Acc_PunchSoft; 
AxAbs_2.Jerk :=3600000;
AxAbs_2.BufferMode :=MC_BUFFER_MODE.Aborting;
AxAbs_2.Dir := MC_DIRECTION.mcPositive;
END_ACTION

ACTION act_45_PunchSoft_PunchB1:
AxAbs_0.Position :=360 - TCP.iPSP1_deg;		
AxAbs_0.Speed :=TCP.iPunchSpeed_Max*6;
AxAbs_0.Acc := AxAbs_0.Dcc :=Def.Acc_PunchSoft; 
AxAbs_0.Jerk :=3600000;
AxAbs_0.BufferMode :=MC_BUFFER_MODE.BlendingLow;
AxAbs_0.Dir := MC_DIRECTION.mcNegative;
END_ACTION

ACTION act_46_PunchSoft_PunchB2:
AxAbs_1.Position :=360 - TCP.iPSP2_deg;		
AxAbs_1.Speed :=TCP.iPunchSpeed*6;
AxAbs_1.Acc := AxAbs_1.Dcc :=Def.Acc_PunchSoft; 
AxAbs_1.Jerk :=3600000;
AxAbs_1.BufferMode :=MC_BUFFER_MODE.BlendingLow;
AxAbs_1.Dir := MC_DIRECTION.mcNegative;
END_ACTION

ACTION act_47_PunchSoft_PunchB3:
AxAbs_2.Position :=TCP.iPOP_deg;		
AxAbs_2.Speed :=TCP.iPunchSpeed_Max*6;
AxAbs_2.Acc := AxAbs_2.Dcc :=Def.Acc_PunchSoft; 
AxAbs_2.Jerk :=3600000;
AxAbs_2.BufferMode :=MC_BUFFER_MODE.Aborting;
AxAbs_2.Dir := MC_DIRECTION.mcNegative;
END_ACTION

ACTION act_7_GoPTE:
// 7 - GoPTE
AxAbs_0.Position :=0;		
AxAbs_0.Speed :=Def.Speed_Go_PTE*6;
AxAbs_0.Acc := AxAbs_0.Dcc :=Def.Acc_Go_PTE; 
AxAbs_0.Jerk :=3600000;
AxAbs_0.BufferMode :=MC_BUFFER_MODE.Aborting;
AxAbs_0.Dir := MC_DIRECTION.mcNegative;

IF ActPos>180 THEN
	AxAbs_0.Dir := MC_DIRECTION.mcPositive;
	AxAbs_0.Position :=360;
END_IF
END_ACTION

ACTION act_Jump_To_PTE:
IF mGoPTE OR wModeSel<>actModeSet THEN
	bFreeMark :=false; //复位自由打标模式信号
	iStep :=7;//Back to PTE
END_IF
END_ACTION

END_PROGRAM

// Device/Application/prTestFunction
PROGRAM prTestFunction
VAR
	FB_Toggle_TestOn :FB_Toggle;
	iTest_Counter :INT;
	iTest_Step :INT;
	iStep_Counter :INT :=0;
	iTest_Punch_Mode AT %MW1601:WORD;
	iTest_Punch_POP_mm AT %MD1602:REAL :=9;
	iTest_Punch_Delay AT %MW1603:INT :=600;
	FB_HeightToAngle_Pop :FB_HeightToAngle;
	FB_Toggle_bTest_iPOP :FB_Toggle;
END_VAR


FB_Toggle_TestOn(Key:= bTest_OnOff , Set:= , Reset:= , Out=> bTest);
FB_Toggle_bTest_iPOP(Key:= bTest_iPOP , Set:= , Reset:= NOT bTest, Out=> bTest_GoPOP);

IF bTest THEN
	Tcp.iPOP_mm :=iTest_Punch_POP_mm;
	FB_HeightToAngle_Pop(HeightMM:= iTest_Punch_POP_mm, AngleDeg=>Tcp.iPOP_deg );
	wModeSel:= iTest_Punch_Mode;
ELSE
	iTest_Step :=0;
	iTest_Counter := iStep_Counter :=0;
END_IF

CASE iTest_Step OF
	0:
//		bTest_iPunch :=bTest_iPOP :=FALSE;
		bTest_iPunch :=FALSE;
		IF bTest AND bTest_GoPOP THEN
			iTest_Step:=10;
		END_IF
	10:
		act_Jump_To_PTE();
		iStep_Counter :=iStep_Counter+1;
		IF iStep_Counter>100 THEN
//			bTest_iPOP :=TRUE;
			iStep_Counter :=0;
			iTest_Step:=20;
		END_IF
	20:
		act_Jump_To_PTE();
		iStep_Counter :=iStep_Counter+1;
		IF iStep_Counter>200 THEN
//			bTest_iPOP :=FALSE;
			iStep_Counter :=0;
			iTest_Step:=30;
		END_IF

	30:	
		act_Jump_To_PTE();
		iStep_Counter :=iStep_Counter+1;
		IF iStep_Counter>200 THEN
			bTest_iPunch :=TRUE;
			iStep_Counter :=0;
			iTest_Step:=40;
		END_IF
		
	40:
		act_Jump_To_PTE();
		iStep_Counter :=iStep_Counter+1;
		IF iStep_Counter>3 THEN
			bTest_iPunch :=FALSE;
			iStep_Counter :=0;
			iTest_Step:=50;
		END_IF
	
	50:
		act_Jump_To_PTE();	
		IF bTest AND qbReadyFeed AND NOT bTest_iPunch THEN	
			iStep_Counter :=iStep_Counter+1;
			IF iStep_Counter>iTest_Punch_Delay THEN
				bTest_iPunch := TRUE;
				iStep_Counter :=0;
				iTest_Step:=40;
			END_IF
		END_IF
	
END_CASE

ACTION act_Jump_To_PTE:
IF NOT bTest_GoPOP  THEN
	iStep_Counter :=0;
	iTest_Step :=0;//Back to PTE
END_IF
END_ACTION

END_PROGRAM

// Device/Application/FunctionBlock/FB_Toggle
FUNCTION_BLOCK FB_Toggle
VAR_INPUT
    Key   : BOOL;  // 按键输入
    Set   : BOOL;  // 置位
    Reset : BOOL;  // 复位
END_VAR
VAR_OUTPUT
    Out   : BOOL;  // 输出状态
END_VAR
VAR
    prevKey : BOOL; // 上一次按键状态
END_VAR

// ------------------- 主逻辑 -------------------

// Set 优先级最高
IF Set THEN
    Out := TRUE;
ELSIF Reset THEN
    Out := FALSE;
ELSE
    // 检测按键上升沿
    IF (Key = TRUE) AND (prevKey = FALSE) THEN
        Out := NOT Out; // 翻转
    END_IF
END_IF

// 更新上一次按键状态
prevKey := Key;

END_FUNCTION_BLOCK

// Device/Application/FunctionBlock/FB_HeightToAngle
FUNCTION_BLOCK FB_HeightToAngle
VAR_INPUT
    HeightMM : REAL; (* 输入高度，单位mm，范围 0~32 *)
END_VAR
VAR_OUTPUT
    AngleDeg : REAL; (* 输出角度，单位°，范围 0~180 *)
END_VAR
VAR
    RR      : REAL := 16.0;   (* 曲柄半径 *)
    L      : REAL := 220.0;  (* 连杆长度 *)
    y_min  : REAL;
    Y      : REAL;
    k      : REAL;
	xll		:REAL;
END_VAR

IF HeightMM>2*RR THEN
	HeightMM :=2*RR;
ELSE
	IF HeightMM<0 THEN
		HeightMM :=0;
	END_IF
END_IF

(* 基准高度：180°最低点 *)
y_min := -RR + L;

(* 滑块绝对高度 *)
xll := HeightMM + y_min;

(* 计算 cos(theta) *)
k := (xll*xll + RR*RR - L*L) / (2.0 * xll * RR);

(* 限制 k 在 -1~1 防止浮点误差 *)
IF k > 1.0 THEN
    k := 1.0;
ELSIF k < -1.0 THEN
    k := -1.0;
END_IF

(* 0 mm 对应 180°，32 mm 对应 0° *)
AngleDeg := ACOS(k) * 180.0 / 3.14159265359;

END_FUNCTION_BLOCK

// Device/Application/DebugMode
PROGRAM DebugMode
VAR
	// ---------- HMI 输入信号 ----------
	bMCHomeExe          : BOOL;

	nStep               : INT;
	iCounter            : INT; 
	iDebugErr           : INT;
	iRetryCount         : INT;
	
	trHome              : R_TRIG;
    trMovePos           : R_TRIG;
    trMoveNeg           : R_TRIG;
	
	fbHome              : MC_Home;
END_VAR

// ---------------- 上升沿检测 ----------------
trHome(CLK := bHomeBtn);
trMovePos(CLK := bMovePosBtn);
trMoveNeg(CLK := bMoveNegBtn);
act_SetHome();

// ---------------- 安全条件监测 ----------------
// 若调试模式关闭或使能关闭 -> 立即复位到初始状态
IF (NOT bDebugModeEnable) OR (NOT bDebugEnableBtn) THEN
    // 状态初始化
    bDebugEnable :=FALSE;
	bMCHomeExe := FALSE;
    iCounter :=0;
    iDebugErr :=0;
    nStep := 0;
	iRetryCount :=0;
    RETURN; // 强制退出本周期，防止执行后续逻辑
END_IF

// ---------------- 主控制逻辑 ----------------
CASE nStep OF

    0: // 等待调试模式 + 伺服使能
		IF bDebugEnableBtn AND (iRetryCount < 5) THEN
			bDebugEnable :=TRUE;
			nStep :=1;
		ELSIF iRetryCount >= 5 THEN
			iDebugErr.0 := TRUE;
		END_IF
	1:
		IF AxisVars.Axis0.AxisMotionState.ServoEnabled AND NOT MC_POWER0.Error THEN
			nStep :=10;
		ELSIF MC_POWER0.Error THEN
			bDebugEnable :=FALSE;
			iCounter :=0;
			nStep :=2;
		END_IF
	2:
		iCounter := iCounter + 1;
        IF iCounter >= 200 THEN
            iCounter := 0;
            nStep := 3;            // 开始执行Reset
        END_IF
	3:
		iCounter := iCounter + 1;
		IF iCounter < 100 THEN
			bReset :=TRUE;
		ELSIF (iCounter >= 100) AND (iCounter < 200) THEN
			bReset :=FALSE;
		ELSIF iCounter >= 200 THEN
			iRetryCount := iRetryCount + 1;
			iCounter := 0;
            nStep := 0;
        END_IF
    10: // 等待操作命令
		AxAbs_0.bExe := bMCHomeExe := FALSE;
		iCounter := 0;
        IF trHome.Q THEN
            nStep := 20;
			iDebugErr := 0;
        ELSIF trMovePos.Q THEN
            nStep := 30;
			iDebugErr := 0;
        ELSIF trMoveNeg.Q THEN
            nStep := 40;
			iDebugErr := 0;
        END_IF

    20: // -------- 回原操作 --------
        bMCHomeExe :=TRUE;
        IF fbHome.Done THEN
            bMCHomeExe := FALSE;
            nStep := 10;
        ELSIF fbHome.Error THEN
			bMCHomeExe := FALSE;
            iDebugErr.1 := TRUE;
            nStep := 10;
        END_IF

    30: // -------- 正向移动 --------
        act_MovePositive();
		AxAbs_0.bExe :=TRUE;
		IF MC_Abs_0.Active THEN
			nStep :=35;
		END_IF		
		
	35:	
		IF MC_Abs_0.Done THEN
			AxAbs_0.bExe :=FALSE;
			nStep :=10;		
		ELSIF MC_Abs_0.Error THEN
			iDebugErr.2 := TRUE;
			AxAbs_0.bExe :=FALSE;
            nStep := 10;
		END_IF		

    40: // -------- 反向移动 --------
        act_MoveNegative();
		AxAbs_0.bExe :=TRUE;
		IF MC_Abs_0.Active THEN
			nStep :=45;
		END_IF

	45:	
		IF MC_Abs_0.Done THEN
			AxAbs_0.bExe :=FALSE;
			nStep :=10;			
		ELSIF MC_Abs_0.Error THEN
			iDebugErr.2 := TRUE;
			AxAbs_0.bExe :=FALSE;
            nStep := 10;
		END_IF

END_CASE;

ACTION act_MoveNegative:

AxAbs_0.Position :=rDebug_TargPos;		
AxAbs_0.Speed :=300*6;
AxAbs_0.Acc := AxAbs_0.Dcc :=36000; 
AxAbs_0.Jerk :=3600000;
AxAbs_0.BufferMode :=MC_BUFFER_MODE.Aborting;
AxAbs_0.Dir := MC_DIRECTION.mcNegative;
END_ACTION

ACTION act_MovePositive:

AxAbs_0.Position :=rDebug_TargPos;		
AxAbs_0.Speed :=300*6;
AxAbs_0.Acc := AxAbs_0.Dcc :=36000; 
AxAbs_0.Jerk :=3600000;
AxAbs_0.BufferMode :=MC_BUFFER_MODE.Aborting;
AxAbs_0.Dir := MC_DIRECTION.mcPositive;
END_ACTION

ACTION act_SetHome:
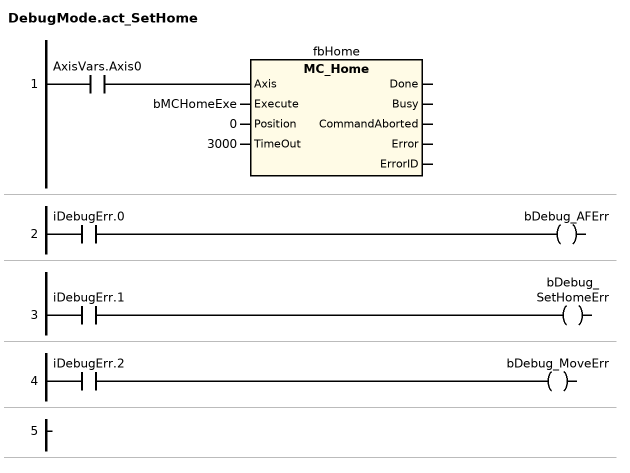
// NETWORK 1
fbHome(Axis := AxisVars.Axis0, Execute := bMCHomeExe, Position := 0, TimeOut := 3000); // MC_Home

// NETWORK 2
bDebug_AFErr := iDebugErr.0;

// NETWORK 3
bDebug_SetHomeErr := iDebugErr.1;

// NETWORK 4
bDebug_MoveErr := iDebugErr.2;

// NETWORK 5
END_ACTION

END_PROGRAM

// Device/Application/ModbusTCP_MasterPRG
(* Auto-Generated Code by 'Modbus Configurator'.
 * DO NOT MODIFY HERE!
 * Changes will be overwritten.
 * If modification is required create a copy of this object. *)
PROGRAM ModbusTCP_MasterPRG
VAR
DoModbusRWList :ARRAY[0..1] OF BOOL;
  TONList : ARRAY[0..1] OF TON;
  NowModbusRWIndex : INT;
  Cycle : INT;  Modbus_TCP_Set1 : Modbus_TCP_Set;
  IP1 : ARRAY [0..3] OF BYTE := [172, 16, 10, 11];
  ModbusRead1 : Modbus_TCP_Read;
  ModbusWrite2 : Modbus_TCP_Write;
  i : INT;
END_VAR

(* Auto-Generated Code by 'Modbus Configurator'.
 * DO NOT MODIFY HERE!
 * Changes will be overwritten.
 * If modification is required create a copy of this object. *)

//Slave1 ModbusTCP connect 172.16.10.11
Modbus_TCP_Set1(Execute:= TRUE, Chn:= COM_LIB.ModbusTcp_CHN_TYPE.ETH, IP:=IP1, 
    Done =>, Socket =>, Error =>, ErrorID =>ModbusTCP_MasterVars.Slave1TCPSetErrorId);

TONList[0](IN:=TRUE, PT:= T#100MS);
TONList[1](IN:=TRUE, PT:= T#100MS);



FOR Cycle := 0 TO 1  DO
  IF NOT DoModbusRWList[NowModbusRWIndex] THEN
    IF TONList[NowModbusRWIndex-0].Q THEN
      TONList[NowModbusRWIndex-0](IN:=FALSE);
      DoModbusRWList[NowModbusRWIndex] := TRUE;
      EXIT;
    ELSE
      NowModbusRWIndex := NowModbusRWIndex + 1;
      NowModbusRWIndex := NowModbusRWIndex MOD 2;
    END_IF
  ELSE
    EXIT;
  END_IF
END_FOR


//Slave1 ModbusTCP Id1 ReadHolding ModbusRead1
IF DoModbusRWList[0] THEN
  ModbusRead1(Execute:= DoModbusRWList[0], Chn:= COM_LIB.ModbusTcp_CHN_TYPE.ETH, Socket:=Modbus_TCP_Set1.Socket, ID:= 2, 
    AddrType:= COM_LIB.Modbus_READ_REG_TYPE.HoldingReg, Addr:= 0, Num:= 10, 
    TimeOut:= 1000, pByteBuf:= ADR(ModbusTCP_MasterVars.Slave1Id1RBuff), ByteBufSize:= 20,
    Done =>, Busy =>, Error =>, ErrorID =>ModbusTCP_MasterVars.Slave1Id1RErrorId);

  IF ModbusRead1.Done THEN
    Tcp.intermediate_iPOP_mm := ModbusTCP_MasterVars.Slave1Id1RBuff[0];
    Tcp.intermediate_iReady_mm := ModbusTCP_MasterVars.Slave1Id1RBuff[1];
    Tcp.intermediate_iPUP_mm := ModbusTCP_MasterVars.Slave1Id1RBuff[2];
    Tcp.intermediate_iDelayTime_ms := ModbusTCP_MasterVars.Slave1Id1RBuff[3];
    Tcp.intermediate_iPSP2_mm := ModbusTCP_MasterVars.Slave1Id1RBuff[4];
    Tcp.intermediate_iPSP1_mm := ModbusTCP_MasterVars.Slave1Id1RBuff[5];
    Tcp.intermediate_iPunchSpeed := ModbusTCP_MasterVars.Slave1Id1RBuff[6];
    Tcp.intermediate_iPunchSpeed_Max := ModbusTCP_MasterVars.Slave1Id1RBuff[7];

  END_IF

  IF ModbusRead1.Done OR ModbusRead1.Error THEN
    ModbusRead1(Execute:= FALSE);
    DoModbusRWList[0] := FALSE;
    NowModbusRWIndex := NowModbusRWIndex + 1;
    NowModbusRWIndex := NowModbusRWIndex MOD 2;
  END_IF
END_IF

//Slave1 ModbusTCP Id2 WriteMultipleHolding ModbusWrite2
IF DoModbusRWList[1] THEN
  ModbusTCP_MasterVars.Slave1Id2WBuff[6].0 := bIdle;
  ModbusWrite2(Execute:= DoModbusRWList[1], Chn:= COM_LIB.ModbusTcp_CHN_TYPE.ETH,  Socket:=Modbus_TCP_Set1.Socket, ID:= 2, 
    AddrType:= COM_LIB.Modbus_WRITE_REG_TYPE.MultiRegisters, Addr:= 20, Num:= 10, 
    TimeOut:= 1000, pByteBuf:= ADR(ModbusTCP_MasterVars.Slave1Id2WBuff), ByteBufSize:= 20,
    Done =>, Busy =>, Error =>, ErrorID =>ModbusTCP_MasterVars.Slave1Id2WErrorId);

  IF ModbusWrite2.Done OR ModbusWrite2.Error THEN
    ModbusWrite2(Execute:= FALSE);
    DoModbusRWList[1] := FALSE;
    NowModbusRWIndex := NowModbusRWIndex + 1;
    NowModbusRWIndex := NowModbusRWIndex MOD 2;
  END_IF
END_IF

END_PROGRAM

// Device/Application/MosbusTcp/prHMI
PROGRAM prHMI
VAR
	Vel_Gain AT %MD1000:REAL;

	iPTE_mm AT %MW1200:WORD;
	iPOP_mm AT %MW1202:WORD;
	iPUP_mm AT %MW1204:WORD;
	iReady_mm AT %MW1206:WORD;
	iDelayTime_ms AT %MW1208:WORD;
	iPunchSpeed_Max AT %MW1210:WORD;
	iPSP1_mm AT %MW1212:WORD;
	iPunchSpeed AT %MW1214:WORD;
	iPSP2_mm AT %MW1216:WORD;
	wMode_hmi AT %MW1218:WORD;
	wActPos AT %MD1220:REAL;
	wPunHeight_mm AT %MW1224:WORD;
	wStep AT %MW1226:WORD;
	iMotorTemperature AT %MW1228:INT;
	wCommuanomaly AT %MW1230:WORD;
	wSetPosExe AT %MW1232:WORD;	
	wdSetPosValue AT %MD1234:REAL;
	
	
	FB_CrankSliderHeight_1 :FB_CrankSliderHeight;

	wI0 AT %MW1500:BYTE;
	wQ20 AT %MW1501:WORD;
	
	Set_RetaParam AT %MD3600:REAL;
	
END_VAR

wI0  := %IB0;
wQ20 := %QW10;

iPTE_mm := TO_WORD(Tcp.iPTE_mm *100);
iPOP_mm := TO_WORD(Tcp.iPOP_mm *100);
iPUP_mm := TO_WORD(Tcp.iPUP_mm *100);
iReady_mm := TO_WORD(Tcp.iReady_mm *100);
iDelayTime_ms := TO_WORD(Tcp.iDelayTime_ms);
iPunchSpeed_Max := TO_WORD(Tcp.intermediate_iPunchSpeed_Max*10);
iPSP1_mm := TO_WORD(Tcp.iPSP1_mm *100);
iPunchSpeed := TO_WORD(Tcp.iPunchSpeed *10);
iPSP2_mm := TO_WORD(Tcp.iPSP2_mm *100);
wActPos := DINT_TO_REAL(LREAL_TO_DINT(ActPos * 100)) / 100;
wPunHeight_mm := TO_WORD(PunHeight *100);
wStep := TO_WORD(iStep);

wMode_hmi := wModeSel;
wCommuanomaly.0 := Tcp.bError;

bSetPosExe := wSetPosExe.0;
SetPosValue := INT_TO_LREAL(REAL_TO_INT(wdSetPosValue * 100)) / 100;

FB_CrankSliderHeight_1(AngleDeg:= TO_REAL(ActPos), HeightMM=> PunHeight);

END_PROGRAM

// Device/Application/FunctionBlock/FB_CrankSliderHeight
FUNCTION_BLOCK FB_CrankSliderHeight
VAR_INPUT
    AngleDeg : REAL; (* 输入曲柄角度，单位° *)
END_VAR
VAR_OUTPUT
    HeightMM : REAL; (* 输出滑块高度，单位mm *)
END_VAR
VAR
    RR       : REAL := 16.0;   (* 曲柄半径mm *)
    L       : REAL := 220.0;  (* 连杆长度mm *)
    angleRad: REAL;
END_VAR


angleRad := AngleDeg * 3.14159265359 / 180.0;

HeightMM := RR
          + RR * COS(angleRad)
          + SQRT(L*L - (RR * SIN(angleRad)) * (RR * SIN(angleRad)))
          - L;

END_FUNCTION_BLOCK

// Device/Application/prCoolFan
//冷却风扇设定打开
PROGRAM prCoolFan 
VAR
	iTimerCounter :UDINT :=0;
END_VAR

IF bAFOn AND iStep>15 OR (TO_INT(iMotorTemp*0.1) > Def.CoolFan_OnTemp)  THEN
	qbFan :=TRUE;
	iTimerCounter :=0;
ELSE
	iTimerCounter := iTimerCounter +1;
	IF TO_INT(iTimerCounter*0.01) > Def.CoolFan_Toff THEN
		iTimerCounter := TO_UDINT(100*(Def.CoolFan_Toff+10));
		qbFan :=FALSE;
	END_IF
END_IF

END_PROGRAM

// Device/Application/MosbusTcp/prHMI_Error
PROGRAM prHMI_Error
VAR
	
(* 驱动器报警输入字 *)
DrvAlarmCode AT %IW16: UINT;  //真实 Errorcode，取PDO参数低8位

(* PLC 内部报警 *)
PlcAlarm_OverTemp : BOOL; 
PlcAlarm_EStop    : BOOL; 

(* 最终报警数组，对应 HMI 1400~1500 地址 *)
HmiAlarm AT %MW1400 : ARRAY [0..99] OF WORD; 
AlarmBits : ARRAY[0..99] OF BOOL; 

i : INT;
	
END_VAR
(* 报警号映射表，对应 Er034 ~ Er160 *)
VAR
    DrvAlarmMap : ARRAY[0..36] OF BYTE := [
		34, 35, 49, 50, 51, 53, 54, 55, 56, 57, 58, 59, 60, 61, 62, 63, 66, 67, 68, 
		69, 70, 81, 82, 83, 84, 89, 90, 109, 110, 111, 122, 132, 144, 145, 146, 147, 160
    ];
END_VAR

(* 1. 清除所有报警位 *)
FOR i := 0 TO 99 DO
    AlarmBits[i] := FALSE;
END_FOR

(* 2. 判断驱动器报警码 *)
FOR i := 0 TO 36 DO
    IF DrvAlarmCode = DrvAlarmMap[i] THEN
        AlarmBits[i] := TRUE;   (* 比如 i=0 对应 Er034 *)
    END_IF
END_FOR

(* 3. PLC 内部报警 *)
//AlarmBits[40] := TCP.bError;
AlarmBits[41] := PlcAlarm_OverTemp;
AlarmBits[42] := PlcAlarm_EStop;
AlarmBits[51] := bDebug_AFErr;
AlarmBits[52] := bDebug_MoveErr;
AlarmBits[53] := bDebug_SetHomeErr;

(* 4. 写入到 HMI Modbus 地址区 *)
FOR i := 0 TO 99 DO
    IF AlarmBits[i] THEN
        HmiAlarm[i] := 1;
    ELSE
        HmiAlarm[i] := 0;
    END_IF
END_FOR

(* 给数控系统报警 *)
IF DrvAlarmCode<>0 THEN
	bDriveError := TRUE; 		
ELSE	
	bDriveError := FALSE; 		
END_IF

END_PROGRAM

// Device/Application/SDO_test
PROGRAM SDO_test
VAR
	
	tBlink : TON;
    LedOut : BOOL;
	SDO_SlaveNum :BYTE;
	
	EtherCAT_SDO_Read_1: EtherCAT_SDO_Read;
	EtherCAT_SDO_DATA1: EtherCAT_SDO_DATA;
	EtherCAT_Status_Update_1: EtherCAT_Status_Update;
	EtherCAT_TYPE_STRUCT1: EtherCAT_TYPE_STRUCT	;
	
	read: BOOL;
END_VAR

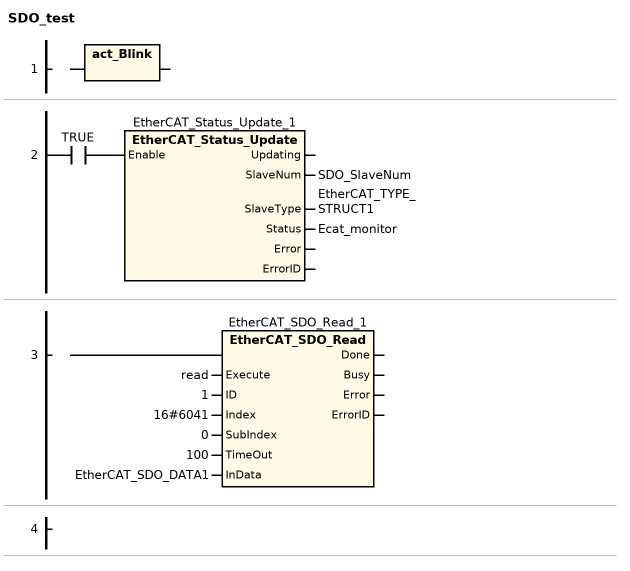
// NETWORK 1
act_Blink();

// NETWORK 2
EtherCAT_Status_Update_1(
    Enable := TRUE,
    SlaveNum => SDO_SlaveNum,
    SlaveType => EtherCAT_TYPE_STRUCT1,
    Status => Ecat_monitor); // EtherCAT_Status_Update

// NETWORK 3
EtherCAT_SDO_Read_1(
    Execute := read,
    ID := 1,
    Index := 16#6041,
    SubIndex := 0,
    TimeOut := 100,
    InData := EtherCAT_SDO_DATA1); // EtherCAT_SDO_Read

// NETWORK 4

ACTION act_Blink:
(* 2s呼吸灯 占空比50%*)
tBlink(IN:=TRUE, PT:=T#1S);    // 定时 1s
IF tBlink.Q THEN
    LedOut := NOT LedOut;      // 翻转输出
    tBlink(IN:=FALSE);         // 重置定时器
END_IF;
END_ACTION

END_PROGRAM

// Device/Application/prIOsetting_test
PROGRAM prIOsetting_test
VAR
	R_TRIG_0: R_TRIG;
	R_TRIG_1: R_TRIG;
	FB_Toggle_0: FB_Toggle;
	bx: BOOL;
	FB_Toggle_1: FB_Toggle;
	FB_Toggle_2: FB_Toggle;
	FB_Toggle_AF: FB_Toggle;
	mModeSel :WORD;
	bStaticState: BOOL;
END_VAR

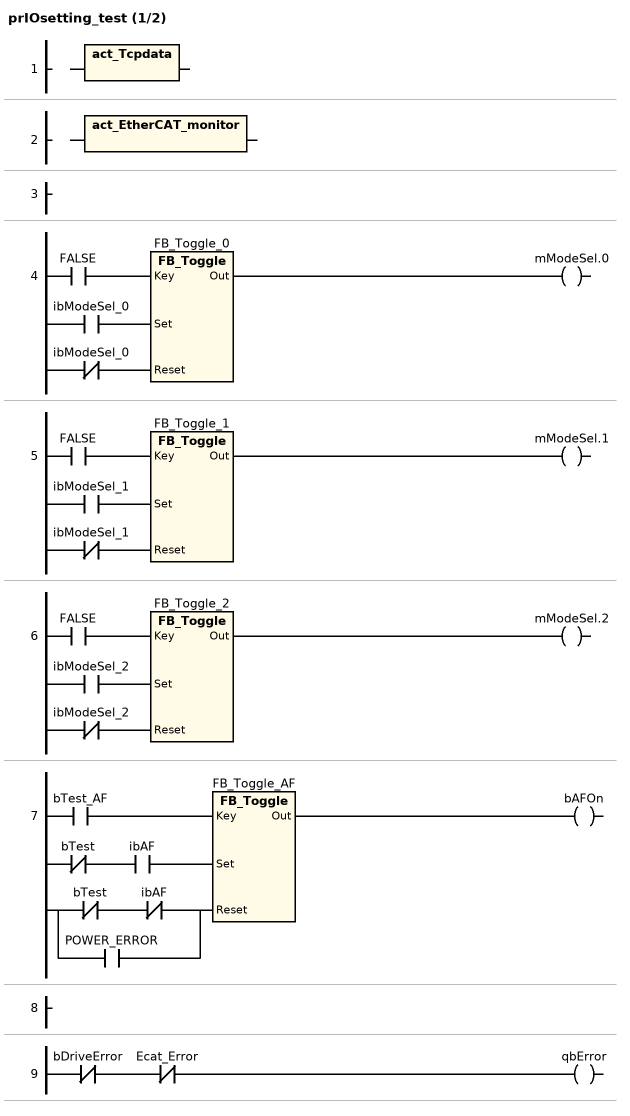
// NETWORK 1
act_Tcpdata();

// NETWORK 2
act_EtherCAT_monitor();

// NETWORK 3

// NETWORK 4
FB_Toggle_0(Key := FALSE, Set := ibModeSel_0, Reset := NOT ibModeSel_0); // FB_Toggle
mModeSel.0 := FB_Toggle_0.Out;

// NETWORK 5
FB_Toggle_1(Key := FALSE, Set := ibModeSel_1, Reset := NOT ibModeSel_1); // FB_Toggle
mModeSel.1 := FB_Toggle_1.Out;

// NETWORK 6
FB_Toggle_2(Key := FALSE, Set := ibModeSel_2, Reset := NOT ibModeSel_2); // FB_Toggle
mModeSel.2 := FB_Toggle_2.Out;

// NETWORK 7
FB_Toggle_AF(Key := bTest_AF, Set := NOT bTest AND ibAF, Reset := NOT bTest AND NOT ibAF OR POWER_ERROR); // FB_Toggle
bAFOn := FB_Toggle_AF.Out;

// NETWORK 8

// NETWORK 9
qbError := NOT bDriveError AND NOT Ecat_Error;

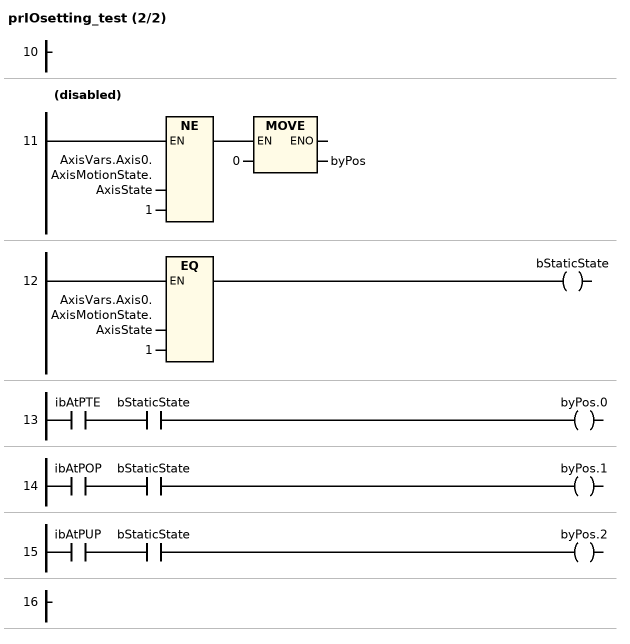
// NETWORK 10

// NETWORK 11 (disabled)
// IF AxisVars.Axis0.AxisMotionState.AxisState <> 1 THEN byPos := 0; END_IF

// NETWORK 12
bStaticState := AxisVars.Axis0.AxisMotionState.AxisState = 1;

// NETWORK 13
byPos.0 := ibAtPTE AND bStaticState;

// NETWORK 14
byPos.1 := ibAtPOP AND bStaticState;

// NETWORK 15
byPos.2 := ibAtPUP AND bStaticState;

// NETWORK 16

ACTION act_EtherCAT_monitor:
IF Ecat_monitor <> 0 THEN
    Ecat_Error := FALSE;
ELSE
    Ecat_Error := TRUE;
END_IF
END_ACTION

ACTION act_Tcpdata:
IF bTest THEN
	Tcp.iPTE_mm := 32;
//	Tcp.iPOP_mm :=16.1 ;
	Tcp.iPUP_mm :=3.1;
	Tcp.iReady_mm :=30;
	Tcp.iDelayTime_ms :=1000;
	Tcp.iPunchSpeed_Max :=400;
	Tcp.iSoftPunch :=0;
	Tcp.iPSP1_mm := 6.1;
	Tcp.iFormMode :=0;
	Tcp.iPSP2_mm :=0.1;
	Tcp.iPunchSpeed :=100;	
ELSE
	wModeSel :=mModeSel;	
END_IF
END_ACTION

END_PROGRAM

// Device/Application/MosbusTcp/prModusTcp_Fanuc
PROGRAM prModusTcp_Fanuc
VAR
	iStep :int;
	Modbus_TCP_Set_0: Modbus_TCP_Set;
	bModbusSet :BOOL;
	Modbus_TCP_Read_0 :Modbus_TCP_Read;
	ipFanuc : ARRAY [0..3] OF BYTE:=[172,16,10,11];
	iCounter :INT;
	bRead :BOOL;
	tcpsocket:BYTE;
	rdata:ARRAY[0..9] OF WORD;
//	bModbusSet_Error :BOOL;
//	bModbusRead_Error :BOOL;
//	bModbusWrite_Error :BOOL;	
	Modbus_TCP_Write_0 :Modbus_TCP_Write;
	bWrite :BOOL;
	wdata:ARRAY[0..9] OF WORD;
//	bIdle :BOOL;
	iReady_deg :REAL;//Data_4换模位置 ready 信号区域
		
	FB_HeightToAngle_iPTE :FB_HeightToAngle;
	FB_HeightToAngle_iPOP :FB_HeightToAngle;
	FB_HeightToAngle_iPUP :FB_HeightToAngle;
	FB_HeightToAngle_iReady :FB_HeightToAngle;
	FB_HeightToAngle_iPSP1 :FB_HeightToAngle;
	FB_HeightToAngle_iPSP2 :FB_HeightToAngle;
	FB_BLINK_Idle:FB_BLINK;
END_VAR

(*CASE iStep OF
	0: //准备及初始化
		bModbusSet :=bRead := bWrite := FALSE;
		iCounter:=0;
		IF NOT Modbus_TCP_Set_0.Execute AND NOT Modbus_TCP_Read_0.Execute THEN
			iStep :=10;
		END_IF
	
	10: //建立与从站连接
		bRead := FALSE;
		bWrite := FALSE;
		bModbusSet := TRUE;
		iCounter :=iCounter +1;
		IF iCounter >5 THEN
			IF Modbus_TCP_Set_0.Error  THEN
				iCounter :=0;				
				bModbusSet := FALSE;
				iStep := 20; 
			ELSE
				IF Modbus_TCP_Set_0.Done THEN
					iCounter :=0;
					tcpsocket :=persistentvars.socket :=Modbus_TCP_Set_0.Socket;
					bModbusSet := FALSE;
					iStep :=20;
				END_IF
			END_IF	
		END_IF
		
	20:	//进行一次数据读取
		bRead :=TRUE;
		iCounter :=iCounter +1;
		IF iCounter>2 THEN
			IF 	Modbus_TCP_Read_0.Error OR Modbus_TCP_Set_0.Error THEN
				iStep := iCounter :=0; //报错跳转
			ELSE
				IF 	Modbus_TCP_Read_0.Done THEN
					iCounter :=0; 
					iStep :=30; //解析数据
					bRead :=FALSE;
				END_IF
			END_IF
		END_IF	

	30:	//进行一次数据写入
		bWrite :=TRUE;
		iCounter :=iCounter +1;
		IF iCounter>2 THEN
			IF 	Modbus_TCP_Write_0.Error OR Modbus_TCP_Set_0.Error THEN
				iStep := iCounter :=0; //报错跳转
			ELSE
				IF 	Modbus_TCP_Write_0.Done THEN
					iCounter :=0; 
					iStep :=40; //解析数据
					bWrite := FALSE;
				END_IF
			END_IF
		END_IF			
	
	40: //分析解析Modbus数据
		bRead :=FALSE;
		bWrite := FALSE;
		iCounter :=iCounter +1;
		//处理读入的数据		
		Tcp.iPOP_mm := TO_REAL(rdata[0])*0.1;
		Tcp.iReady_mm := TO_REAL(rdata[1])*0.1;	
	    Tcp.iPUP_mm := TO_REAL(rdata[2])*0.1;
	    Tcp.iDelayTime_ms := TO_UINT(rdata[3]*10);
	    Tcp.iPSP2_mm := TO_REAL(rdata[4])*0.1;
		Tcp.iPSP1_mm := TO_REAL(rdata[5])*0.1;
		Tcp.iPunchSpeed := TO_REAL(rdata[6])*1;
		Tcp.iPunchSpeed_Max := TO_REAL(rdata[7])*1;

		
		IF Tcp.iPTE_mm>20 AND Tcp.iPunchSpeed_Max>100 THEN
			Tcp.iRead_OK :=Tcp.iRead_OK+1;
			IF Tcp.iRead_OK>32000 THEN
				Tcp.iRead_OK :=100;
			END_IF
		ELSE
			Tcp.iRead_OK :=0;	
		END_IF
			
		IF iCounter >1 THEN
			iCounter :=0;
			iStep :=20;
		END_IF
END_CASE

//通讯连接
Modbus_TCP_Set_0(	Execute:= bModbusSet, 	
	Chn:= COM_LIB.ModbusTcp_CHN_TYPE.ETH,	IP:= ipFanuc);

//读从站数据	
Modbus_TCP_Read_0(
	Execute:= bRead, 	
	Chn:= COM_LIB.ModbusTcp_CHN_TYPE.ETH,	Socket:= tcpsocket,	ID:= 1,
	AddrType:= com_lib.Modbus_READ_REG_TYPE.HoldingReg, 
	Addr:= 0, 	Num:= 10,	TimeOut:= 1000, 
	pByteBuf:= ADR(rdata), 	ByteBufSize:= 20, 
	Done=> , 	Busy=> ,	Error=> ,	ErrorID=> );
	
//写从站数据
Modbus_TCP_Write_0(
	Execute:= bWrite, 
	Chn:= COM_LIB.ModbusTcp_CHN_TYPE.ETH, Socket:= tcpsocket, ID:= 1, 
	AddrType:= com_lib.Modbus_WRITE_REG_TYPE.MultiRegisters, 
	Addr:= 20, Num:= 10, TimeOut:= 1000, 
	pByteBuf:= ADR(wdata), ByteBufSize:= 20, 
	Done=> , Busy=> , Error=> , ErrorID=> );


//通讯故障	
IF 	Modbus_TCP_Set_0.Error OR iStep<20 THEN
	bModbusSet_Error :=TRUE;
ELSE
//	IF	Modbus_TCP_Set_0.Execute AND Modbus_TCP_Set_0.Done AND NOT Modbus_TCP_Set_0.Error THEN
		bModbusSet_Error :=FALSE;
//	END_IF 	
END_IF

IF 	Modbus_TCP_Read_0.Error THEN
	bModbusRead_Error :=TRUE;
ELSE
	IF	Modbus_TCP_Read_0.Execute AND Modbus_TCP_Read_0.Done AND NOT Modbus_TCP_Read_0.Error THEN
		bModbusRead_Error :=FALSE;
	END_IF 	
END_IF

IF 	Modbus_TCP_Write_0.Error THEN
	bModbusWrite_Error :=TRUE;
ELSE
	IF	Modbus_TCP_Write_0.Execute AND Modbus_TCP_Write_0.Done AND NOT Modbus_TCP_Write_0.Error THEN
		bModbusWrite_Error :=FALSE;
	END_IF 	
END_IF

//Modbus通讯异常
Tcp.bError := bModbusSet_Error  OR bModbusRead_Error OR bModbusWrite_Error;
FB_BLINK_Idle(Enable:= NOT Tcp.bError, Period:= T#500ms, Q=> bIdle);
IF bIdle THEN
	wdata[6] := 1;
ELSE
	wdata[6] := 0;
END_IF*)
(*
    Tcp.iPOP_mm := TO_REAL(ModbusTCP_MasterVars.Slave1Id1RBuff[0])*0.1;
    Tcp.iReady_mm := TO_REAL(ModbusTCP_MasterVars.Slave1Id1RBuff[1])*0.1;
    Tcp.iPUP_mm := TO_REAL(ModbusTCP_MasterVars.Slave1Id1RBuff[2])*0.1;
    Tcp.iDelayTime_ms := TO_UINT(ModbusTCP_MasterVars.Slave1Id1RBuff[3]*10);
    Tcp.iPSP2_mm := TO_REAL(ModbusTCP_MasterVars.Slave1Id1RBuff[4])*0.1;
    Tcp.iPSP1_mm := TO_REAL(ModbusTCP_MasterVars.Slave1Id1RBuff[5])*0.1;
    Tcp.iPunchSpeed := TO_REAL(ModbusTCP_MasterVars.Slave1Id1RBuff[6]);
    Tcp.iPunchSpeed_Max := TO_REAL(ModbusTCP_MasterVars.Slave1Id1RBuff[7]);
*)
IF NOT bTest THEN
	IF TCP.intermediate_iPunchSpeed_Max>Def.PunchSpeed_Max_Lim THEN 
		Tcp.iPunchSpeed_Max := Def.PunchSpeed_Max_Lim;
	ELSE	
		Tcp.iPunchSpeed_Max := TCP.intermediate_iPunchSpeed_Max;
	END_IF
END_IF

//Modbus通讯异常
Tcp.bError := bModbusSet_Error  OR bModbusRead_Error OR bModbusWrite_Error;
FB_BLINK_Idle(Enable:= NOT Tcp.bError, Period:= T#500MS, Q=> bIdle);

//处理读入的数据
IF NOT bTest THEN
	Tcp.iPOP_mm := TO_REAL(TCP.intermediate_iPOP_mm)*0.1;
	Tcp.iReady_mm := TO_REAL(TCP.intermediate_iReady_mm)*0.1;	
	Tcp.iPUP_mm := TO_REAL(TCP.intermediate_iPUP_mm)*0.1;
	Tcp.iDelayTime_ms := TO_UINT(TCP.intermediate_iDelayTime_ms*10);
	Tcp.iPSP2_mm := TO_REAL(TCP.intermediate_iPSP2_mm)*0.1;
	Tcp.iPSP1_mm := TO_REAL(TCP.intermediate_iPSP1_mm)*0.1;
	Tcp.iPunchSpeed := TO_REAL(TCP.intermediate_iPunchSpeed)*1;
	Tcp.iPunchSpeed_Max := TO_REAL(Tcp.iPunchSpeed_Max)*1;
END_IF

//高度转换角度计算
FB_HeightToAngle_iPTE(HeightMM:= Tcp.iPTE_mm, AngleDeg=> Tcp.iPTE_deg);
FB_HeightToAngle_iPOP(HeightMM:= Tcp.iPOP_mm, AngleDeg=> Tcp.iPOP_deg);
FB_HeightToAngle_iPUP(HeightMM:= Tcp.iPUP_mm, AngleDeg=> Tcp.iPUP_deg);
FB_HeightToAngle_iReady(HeightMM:= Tcp.iReady_mm, AngleDeg=> iReady_deg );
FB_HeightToAngle_iPSP1(HeightMM:= Tcp.iPSP1_mm, AngleDeg=> Tcp.iPSP1_deg);
FB_HeightToAngle_iPSP2(HeightMM:= Tcp.iPSP2_mm, AngleDeg=> Tcp.iPSP2_deg);

//转换到位窗口
Tcp.iReady_deg := 180.0 - iReady_deg;

END_PROGRAM

// Device/Application/FunctionBlock/FB_BLINK
FUNCTION_BLOCK FB_BLINK
VAR_INPUT
	Enable: BOOL;         // 使能信号，TRUE 时启动闪烁
    Period: TIME; // 闪烁周期，如写 1 秒（亮暗各占一半）
END_VAR
VAR_OUTPUT
	Q: BOOL;              // 输出信号，周期性反转
END_VAR
VAR
	Timer: TON;           // 定时器，用于计时
    State: BOOL := FALSE; // 内部状态变量
END_VAR

IF Enable THEN
    // 启动定时器，定时时间为周期的一半
    Timer(IN := NOT Timer.Q, PT := Period / 2);
    
    // 当定时器计时完成时，反转输出状态
    IF Timer.Q THEN
        State := NOT State;
        Timer(IN := FALSE); // 重置定时器
    END_IF;
    
    Q := State; // 输出当前状态
ELSE
    // 未使能时，输出默认值（通常为 FALSE）
    Q := FALSE;
    Timer(IN := FALSE);
    State := FALSE;
END_IF;

END_FUNCTION_BLOCK

// Device/Application/SetHome
PROGRAM SetHome
VAR
	MC_SetPosition_0: MC_SetPosition;
	MC_WriteParameter_0: MC_WriteParameter;
	vvv: AXIS_PARA_ID := AXIS_PARA_ID.WR_DOUBLE_MOTOR_OFFSET;
END_VAR

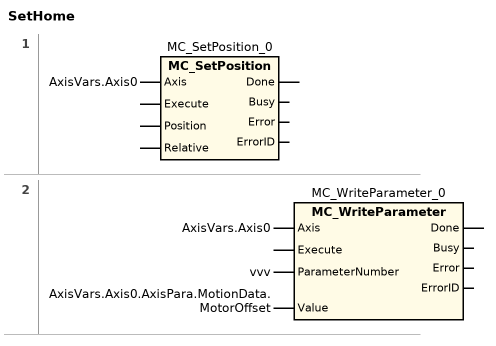
// NETWORK 1
MC_SetPosition_0(Axis := AxisVars.Axis0); // MC_SetPosition

// NETWORK 2
MC_WriteParameter_0(
    Axis := AxisVars.Axis0,
    ParameterNumber := vvv,
    Value := AxisVars.Axis0.AxisPara.MotionData.MotorOffset); // MC_WriteParameter

END_PROGRAM

// Device/Application/SetPosition0
PROGRAM SetPosition0
VAR
	MC_SetPosition_0: MC_SetPosition;
	MC_WriteParameter_0: MC_WriteParameter;
	
	EXsp:BOOL;
	setposition:LREAL :=0;
	relative:BOOL;
	writeP:BOOL:=1;
	
	offsetvalue AT %ML2000:LREAL;
	R_TRIG_0: R_TRIG;
	FB_BLINK_0: FB_BLINK;
	R_TRIG_1: R_TRIG;
	TON_0: TON;
	TOF_0: TOF;
	bSetPosComp: BOOL;
END_VAR

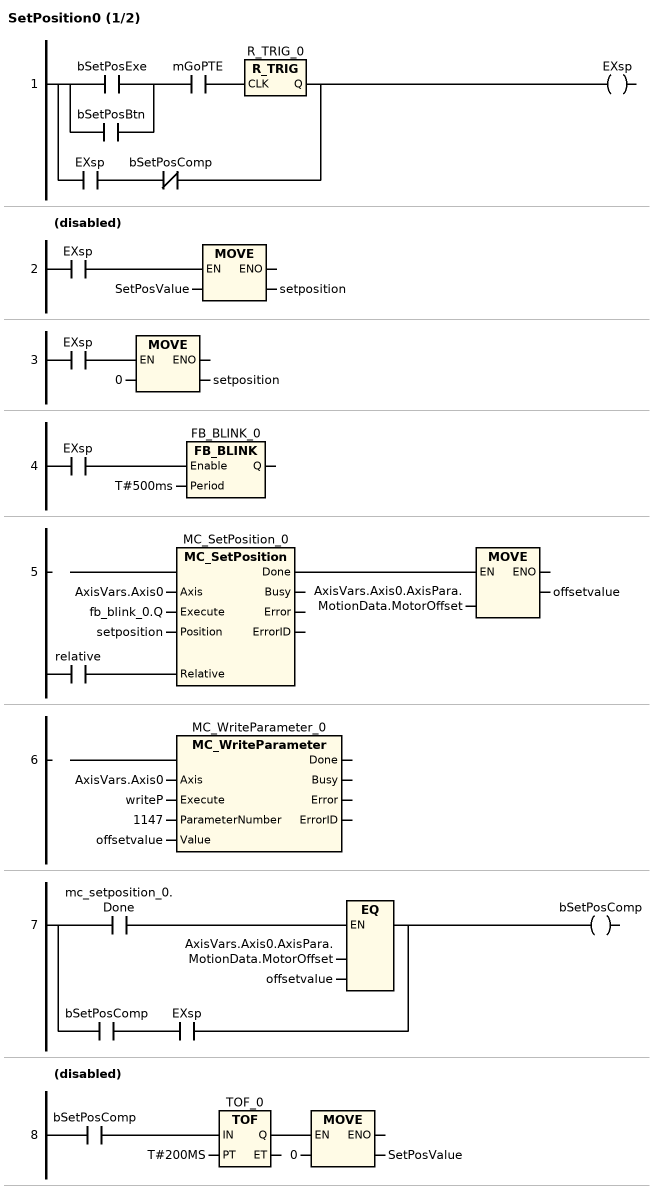
// NETWORK 1
R_TRIG_0(CLK := (bSetPosExe OR bSetPosBtn) AND mGoPTE); // R_TRIG
EXsp := R_TRIG_0.Q OR EXsp AND NOT bSetPosComp;

// NETWORK 2 (disabled)
// IF EXsp THEN setposition := SetPosValue; END_IF

// NETWORK 3
IF EXsp THEN setposition := 0; END_IF

// NETWORK 4
FB_BLINK_0(Enable := EXsp, Period := T#500ms); // FB_BLINK

// NETWORK 5
MC_SetPosition_0(
    Axis := AxisVars.Axis0,
    Execute := fb_blink_0.Q,
    Position := setposition,
    Relative := relative); // MC_SetPosition
IF MC_SetPosition_0.Done THEN offsetvalue := AxisVars.Axis0.AxisPara.MotionData.MotorOffset; END_IF

// NETWORK 6
MC_WriteParameter_0(Axis := AxisVars.Axis0, Execute := writeP, ParameterNumber := 1147, Value := offsetvalue); // MC_WriteParameter

// NETWORK 7
bSetPosComp := mc_setposition_0.Done AND AxisVars.Axis0.AxisPara.MotionData.MotorOffset = offsetvalue OR bSetPosComp AND EXsp;

// NETWORK 8 (disabled)
// TOF_0(IN := bSetPosComp, PT := T#200MS); // TOF
// IF TOF_0.Q THEN SetPosValue := 0; END_IF

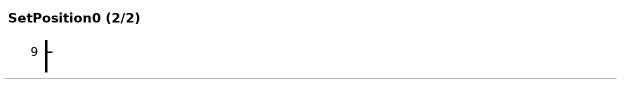
// NETWORK 9

END_PROGRAM

// Device/Application/Test_Crank
PROGRAM Test_Crank
VAR
	FB_CrankSliderHeight_1 :FB_CrankSliderHeight;
	xx :REAL;
	aa :REAL;
	mm :REAL;
	ax :REAL;
	FB_HeightToAngle_1 :FB_HeightToAngle;
END_VAR


FB_HeightToAngle_1(HeightMM:= mm, AngleDeg=> ax);
FB_CrankSliderHeight_1(AngleDeg:= ax, HeightMM=>xx );

END_PROGRAM

// Device/Application/BAK/Punch_PA_1
PROGRAM Punch_PA_1
VAR
	iStep :INT :=0;
	iCounter :INT :=0;
END_VAR

IF NOT bAFOn OR NOT  AxisVars.Axis0.AxisMotionState.ServoEnabled THEN
	iStep := iCounter:=0;
END_IF 

CASE iStep OF
	0://Power Off, reset data
		AxAbs_0.bExe := AxAbs_1.bExe :=AxAbs_2.bExe :=FALSE;
		IF bAFOn AND NOT MC_POWER0.Error AND AxisVars.Axis0.AxisMotionState.ServoEnabled THEN
			iStep :=7;
		END_IF
		
	7://PrePTE
		AxAbs_0.Position :=0;		AxAbs_0.Speed :=100*6;
		AxAbs_0.Acc := AxAbs_0.Dcc :=360000; AxAbs_0.Jerk :=3600000;
		AxAbs_0.BufferMode :=MC_BUFFER_MODE.Aborting;
		AxAbs_0.Dir := MC_DIRECTION.mcNegative;	
		AxAbs_0.bExe := AxAbs_1.bExe :=AxAbs_2.bExe :=FALSE;
		IF ActPos>180 THEN
			AxAbs_0.Dir := MC_DIRECTION.mcPositive;
			AxAbs_0.Position :=360;
		END_IF
		 iCounter:= iCounter +1;
		IF iCounter>100 THEN
			iStep :=10;
			iCounter :=0;
		END_IF	
		
	10://Back to PTE
		AxAbs_0.bExe :=TRUE;
		IF MC_Abs_0.Active THEN
			AxAbs_0.bExe :=FALSE;
		END_IF
		IF MC_Abs_0.Done AND  ibAtPTE THEN
			AxAbs_0.bExe :=FALSE;
			iCounter :=iCounter+1;
			IF iCounter>200 THEN
				iStep :=15;
				iCounter :=0;			
			END_IF
		END_IF
	
	15://Waiting for Switching Mode
		bReady_OnFly :=FALSE;
		CASE wModeSel OF
				0://Punch-A Side
					IF rt_ibGoPOP.Q THEN
						iStep :=20;
					END_IF
					
				1://Wheel
				
			
				2://Forming
	
				
				3://Punch-AB Side
					IF rt_ibGoPOP.Q THEN
						IF ibSoftPun THEN
							iStep :=40;
						ELSE
							iStep :=30;
						END_IF
					END_IF
					
				4://Round 
		END_CASE
		
	20://Punch - Aside - step0 - Go POP
		AxAbs_0.Position :=POP_Pos;		AxAbs_0.Speed :=100*6;
		AxAbs_0.Acc := AxAbs_0.Dcc :=360000; AxAbs_0.Jerk :=3600000;
		AxAbs_0.BufferMode :=MC_BUFFER_MODE.Aborting;
		AxAbs_0.Dir := MC_DIRECTION.mcPositive;	
		AxAbs_0.bExe :=TRUE;
		IF MC_Abs_0.Active THEN
			AxAbs_0.bExe :=FALSE;
		END_IF	
		IF MC_Abs_0.Done THEN
			AxAbs_0.bExe :=FALSE;
			iCounter :=iCounter+1;
			IF iCounter>100 THEN
				iStep :=21;	iCounter :=0;			
			END_IF
		END_IF		
		
	21://Punch - Aside - step1 - Wating Pun-ibPunch
		AxAbs_0.Position :=PUP_Pos;		AxAbs_0.Speed :=Punch_Speed*6;
		AxAbs_0.Acc := AxAbs_0.Dcc :=360000; AxAbs_0.Jerk :=3600000;
		AxAbs_0.BufferMode :=MC_BUFFER_MODE.Aborting;
		AxAbs_0.Dir := MC_DIRECTION.mcPositive;
		AxAbs_0.bExe :=FALSE;	
		IF rt_ibGoPOP.Q OR wModeSel<>0 THEN
			iStep :=7;//Back to PTE
		END_IF
		IF rt_ibPunch.Q THEN
			bReady_OnFly :=FALSE;
			iStep :=22;
		END_IF

		
	22://Punch - Aside - step2
		AxAbs_0.bExe :=TRUE;
		IF MC_Abs_0.Active THEN
			AxAbs_0.bExe :=FALSE;
		END_IF	
		AxAbs_1.Position :=POP_Pos;		AxAbs_1.Speed :=Punch_Speed*6;
		AxAbs_1.Acc := AxAbs_1.Dcc :=360000; AxAbs_1.Jerk :=3600000;
		AxAbs_1.BufferMode :=MC_BUFFER_MODE.Aborting;
		AxAbs_1.Dir := MC_DIRECTION.mcNegative;	
		AxAbs_1.bExe :=FALSE;
		IF MC_Abs_0.Done THEN
			AxAbs_0.bExe :=FALSE;
			iStep :=23;			
		END_IF		
	23://Punch - Aside - step3	
		bReady_OnFly :=TRUE;
		AxAbs_1.bExe :=TRUE;
		IF MC_Abs_1.Done THEN
			AxAbs_1.bExe :=FALSE;
			iStep :=21;			
		END_IF		
	
	
	30://Punch - ABside - step0 - Go POP
		AxAbs_0.Position :=POP_Pos;		AxAbs_0.Speed :=100*6;
		AxAbs_0.Acc := AxAbs_0.Dcc :=360000; AxAbs_0.Jerk :=3600000;
		AxAbs_0.BufferMode :=MC_BUFFER_MODE.Aborting;
		AxAbs_0.Dir := MC_DIRECTION.mcPositive;	
		AxAbs_0.bExe :=TRUE;
		IF MC_Abs_0.Active THEN
			AxAbs_0.bExe :=FALSE;
		END_IF	
		IF MC_Abs_0.Done THEN
			AxAbs_0.bExe :=FALSE;
			iCounter :=iCounter+1;
			IF iCounter>100 THEN
				iStep :=31;	iCounter :=0;			
			END_IF
		END_IF	
		
	31://Punch - ABside - step1 - Wating Pun-ibPunch
		AxAbs_0.Position :=360 - POP_Pos;		AxAbs_0.Speed :=Punch_Speed*6;
		AxAbs_0.Acc := AxAbs_0.Dcc :=360000; AxAbs_0.Jerk :=3600000;
		AxAbs_0.BufferMode :=MC_BUFFER_MODE.Aborting;
		AxAbs_0.Dir := MC_DIRECTION.mcPositive;
		AxAbs_0.bExe :=FALSE;	
		IF rt_ibGoPOP.Q THEN
			iStep :=7;//Back to PTE
		END_IF
		IF rt_ibPunch.Q THEN
			bReady_OnFly :=FALSE;
			iStep :=32;
		END_IF
		
	32://Punch - ABside - step1 - Wating Pun-ibPunch
		AxAbs_0.bExe :=TRUE;
		IF	ActPos>180 THEN
			bReady_OnFly :=TRUE;
		END_IF
		IF rt_ibGoPOP.Q THEN
			iStep :=7;//Back to PTE
		END_IF
		IF MC_Abs_0.Active THEN
			AxAbs_0.bExe :=FALSE;
		END_IF	
		IF MC_Abs_0.Done THEN
			AxAbs_0.bExe :=FALSE;
			iStep :=33;	iCounter :=0;			
		END_IF		
		
	33://Punch - ABside - step1 - Wating Pun-ibPunch
		AxAbs_0.Position :=POP_Pos;		AxAbs_0.Speed :=Punch_Speed*6;
		AxAbs_0.Acc := AxAbs_0.Dcc :=360000; AxAbs_0.Jerk :=3600000;
		AxAbs_0.BufferMode :=MC_BUFFER_MODE.Aborting;
		AxAbs_0.Dir := MC_DIRECTION.mcNegative;
		AxAbs_0.bExe :=FALSE;	
		IF rt_ibGoPOP.Q THEN
			iStep :=7;//Back to PTE
		END_IF
		IF rt_ibPunch.Q THEN
			bReady_OnFly :=FALSE;
			iStep :=34;
		END_IF
		
	34://Punch - ABside - step1 - Wating Pun-ibPunch
		AxAbs_0.bExe :=TRUE;
		IF	ActPos<180 THEN
			bReady_OnFly :=TRUE;
		END_IF	
		IF rt_ibGoPOP.Q THEN
			iStep :=7;//Back to PTE
		END_IF
		IF MC_Abs_0.Active THEN
			AxAbs_0.bExe :=FALSE;
		END_IF	
		IF MC_Abs_0.Done THEN
			AxAbs_0.bExe :=FALSE;
			iStep :=31;	iCounter :=0;			
		END_IF	



	40://Punch - ABside SoftPunch - step0 - Go POP
		AxAbs_0.Position :=POP_Pos;		AxAbs_0.Speed :=100*6;
		AxAbs_0.Acc := AxAbs_0.Dcc :=360000; AxAbs_0.Jerk :=3600000;
		AxAbs_0.BufferMode :=MC_BUFFER_MODE.Aborting;
		AxAbs_0.Dir := MC_DIRECTION.mcPositive;	
		AxAbs_0.bExe :=TRUE;
		IF MC_Abs_0.Active THEN
			AxAbs_0.bExe :=FALSE;
		END_IF	
		IF MC_Abs_0.Done THEN
			AxAbs_0.bExe :=FALSE;
			iCounter :=iCounter+1;
			IF iCounter>100 THEN
				iStep :=41;	iCounter :=0;			
			END_IF
		END_IF	
		
		
		
	41:
		AxAbs_0.Position :=140;		AxAbs_0.Speed :=Punch_Speed*6;
		AxAbs_0.Acc := AxAbs_0.Dcc :=360000; AxAbs_0.Jerk :=3600000;
		AxAbs_0.BufferMode :=MC_BUFFER_MODE.BlendingLow;
		AxAbs_0.Dir := MC_DIRECTION.mcPositive;
		AxAbs_0.bExe :=FALSE;	
		IF rt_ibGoPOP.Q THEN
			iStep :=7;//Back to PTE
		END_IF
		IF rt_ibPunch.Q THEN
			bReady_OnFly :=FALSE;
			iStep :=42;
		END_IF
		
		
		
	42:
		AxAbs_0.bExe :=TRUE;
		AxAbs_1.Position :=180;		AxAbs_1.Speed :=100*6;
		AxAbs_1.Acc := AxAbs_1.Dcc :=360000; AxAbs_1.Jerk :=3600000;
		AxAbs_1.BufferMode :=MC_BUFFER_MODE.BlendingLow;
		AxAbs_1.Dir := MC_DIRECTION.mcPositive;
		AxAbs_1.bExe :=FALSE;
		IF rt_ibGoPOP.Q THEN
			iStep :=7;//Back to PTE
		END_IF
		IF MC_Abs_0.Active THEN
			AxAbs_0.bExe :=FALSE;
		END_IF	
		IF MC_Abs_0.Done THEN
			AxAbs_0.bExe :=FALSE;
			iStep :=43;	iCounter :=0;			
		END_IF	
		
		
		
	43:
		AxAbs_1.bExe :=TRUE;
		AxAbs_2.Position :=360 - POP_Pos;		AxAbs_2.Speed :=Punch_Speed*6;
		AxAbs_2.Acc := AxAbs_2.Dcc :=360000; AxAbs_2.Jerk :=3600000;
		AxAbs_2.BufferMode :=MC_BUFFER_MODE.Aborting;
		AxAbs_2.Dir := MC_DIRECTION.mcPositive;
		AxAbs_2.bExe :=FALSE;
		IF rt_ibGoPOP.Q THEN
			iStep :=7;//Back to PTE
		END_IF
		IF MC_Abs_1.Active THEN
			AxAbs_1.bExe :=FALSE;
		END_IF	
		IF MC_Abs_1.Done THEN
			AxAbs_1.bExe :=FALSE;
			iStep :=44;	iCounter :=0;			
		END_IF
		
		
		
	44:
		AxAbs_2.bExe :=TRUE;
		IF	ActPos>180 THEN
			bReady_OnFly :=TRUE;
		END_IF		
		IF rt_ibGoPOP.Q THEN
			iStep :=7;//Back to PTE
		END_IF
		IF MC_Abs_2.Active THEN
			AxAbs_2.bExe :=FALSE;
		END_IF	
		IF MC_Abs_2.Done THEN
			AxAbs_2.bExe :=FALSE;
			iStep :=45;	iCounter :=0;			
		END_IF
		
		
		
	45:
		AxAbs_0.Position :=220;		AxAbs_0.Speed :=Punch_Speed*6;
		AxAbs_0.Acc := AxAbs_0.Dcc :=360000; AxAbs_0.Jerk :=3600000;
		AxAbs_0.BufferMode :=MC_BUFFER_MODE.BlendingLow;
		AxAbs_0.Dir := MC_DIRECTION.mcNegative;
		AxAbs_0.bExe :=FALSE;	
		IF rt_ibGoPOP.Q THEN
			iStep :=7;//Back to PTE
		END_IF
		IF rt_ibPunch.Q THEN
			bReady_OnFly :=FALSE;
			iStep :=46;
		END_IF
	


	46:
		AxAbs_0.bExe :=TRUE;
		AxAbs_1.Position :=180;		AxAbs_1.Speed :=100*6;
		AxAbs_1.Acc := AxAbs_1.Dcc :=360000; AxAbs_1.Jerk :=3600000;
		AxAbs_1.BufferMode :=MC_BUFFER_MODE.BlendingLow;
		AxAbs_1.Dir := MC_DIRECTION.mcNegative;
		AxAbs_1.bExe :=FALSE;
		IF rt_ibGoPOP.Q THEN
			iStep :=7;//Back to PTE
		END_IF
		IF MC_Abs_0.Active THEN
			AxAbs_0.bExe :=FALSE;
		END_IF	
		IF MC_Abs_0.Done THEN
			AxAbs_0.bExe :=FALSE;
			iStep :=47;	iCounter :=0;			
		END_IF	
		
		
		
	47:
		AxAbs_1.bExe :=TRUE;
		AxAbs_2.Position :=POP_Pos;		AxAbs_2.Speed :=Punch_Speed*6;
		AxAbs_2.Acc := AxAbs_2.Dcc :=360000; AxAbs_2.Jerk :=3600000;
		AxAbs_2.BufferMode :=MC_BUFFER_MODE.Aborting;
		AxAbs_2.Dir := MC_DIRECTION.mcNegative;
		AxAbs_2.bExe :=FALSE;
		IF rt_ibGoPOP.Q THEN
			iStep :=7;//Back to PTE
		END_IF
		IF MC_Abs_1.Active THEN
			AxAbs_1.bExe :=FALSE;
		END_IF	
		IF MC_Abs_1.Done THEN
			AxAbs_1.bExe :=FALSE;
			iStep :=48;	iCounter :=0;			
		END_IF
		
		
		
	48:
		AxAbs_2.bExe :=TRUE;
		IF	ActPos<180 THEN
			bReady_OnFly :=TRUE;
		END_IF		
		IF rt_ibGoPOP.Q THEN
			iStep :=7;//Back to PTE
		END_IF
		IF MC_Abs_2.Active THEN
			AxAbs_2.bExe :=FALSE;
		END_IF	
		IF MC_Abs_2.Done THEN
			AxAbs_2.bExe :=FALSE;
			iStep :=41;	iCounter :=0;			
		END_IF
	
	(*
	20://PreStep for Switching Mode
		AxAbs_0.Position :=80;		AxAbs_0.Speed :=100;
		AxAbs_0.Acc := AxAbs_0.Dcc :=360000; AxAbs_0.Jerk :=3600000;
		AxAbs_0.BufferMode :=MC_BUFFER_MODE.Buffered;
		AxAbs_0.Dir := MC_DIRECTION.mcPositive;	

		AxAbs_0.bExe :=TRUE;
		IF MC_Abs_0.Active THEN
			AxAbs_0.bExe :=FALSE;
		END_IF	
		IF MC_Abs_0.Done THEN
			iStep :=21;
		END_IF	
		
		
	21:
		AxAbs_1.Position :=180;		AxAbs_1.Speed :=20;
		AxAbs_1.Acc := AxAbs_1.Dcc :=360000; AxAbs_1.Jerk :=3600000;
		AxAbs_1.BufferMode :=MC_BUFFER_MODE.Aborting;
		AxAbs_1.Dir := MC_DIRECTION.mcPositive;	
		AxAbs_1.bExe :=TRUE;
		IF MC_Abs_1.Active THEN
			AxAbs_1.bExe :=FALSE;
		END_IF
		IF MC_Abs_1.Done THEN
			iStep :=25;
			AxAbs_1.bExe :=FALSE;
		END_IF
	25:
		iCounter :=iCounter+1;
		IF iCounter>500 THEN
			iStep :=30;
			iCounter :=0;
		END_IF
		
	30://PreStep for Switching Mode
		AxAbs_0.Position :=0;		AxAbs_0.Speed :=100;
		AxAbs_0.Acc := AxAbs_0.Dcc :=360000; AxAbs_0.Jerk :=3600000;
		AxAbs_0.BufferMode :=MC_BUFFER_MODE.Aborting;
		AxAbs_0.Dir := MC_DIRECTION.mcNegative;
		AxAbs_0.bExe :=FALSE;AxAbs_1.bExe :=FALSE;

		iCounter :=iCounter+1;
		IF iCounter>500 THEN
			iStep :=31;
			iCounter :=0;
		END_IF
		
	31:	
		AxAbs_0.bExe :=TRUE;
		IF MC_Abs_0.Active THEN
			AxAbs_0.bExe :=FALSE;
		END_IF		
		IF MC_Abs_0.Done THEN
			iStep :=35;
			AxAbs_0.bExe :=FALSE;		
		END_IF
	35:
		iCounter :=iCounter+1;
		AxAbs_0.BufferMode :=MC_BUFFER_MODE.Buffered;
		AxAbs_1.BufferMode :=MC_BUFFER_MODE.Aborting;
		AxAbs_0.bExe :=FALSE;
		AxAbs_1.bExe :=FALSE;
		IF iCounter>1000 THEN
			iStep :=20;
			iCounter :=0;
		END_IF		
		*)
		
END_CASE

END_PROGRAM

// Device/Application/MosbusTcp/Modbus_Client_Fanuc
PROGRAM Modbus_Client_Fanuc
VAR
	Modbus_TCP_Set_0: Modbus_TCP_Set;
	ip : ARRAY [0..3] OF BYTE:=[172,16,10,11];
	tcpsocket:byte;
	Modbus_TCP_Read_0: Modbus_TCP_Read;
	rdata:ARRAY[0..9] of word;
	busy: BOOL;
	error: BOOL;
	errorid: WORD;
	
	RW	: TON;
	MB_RW	: BOOL:=0;
END_VAR

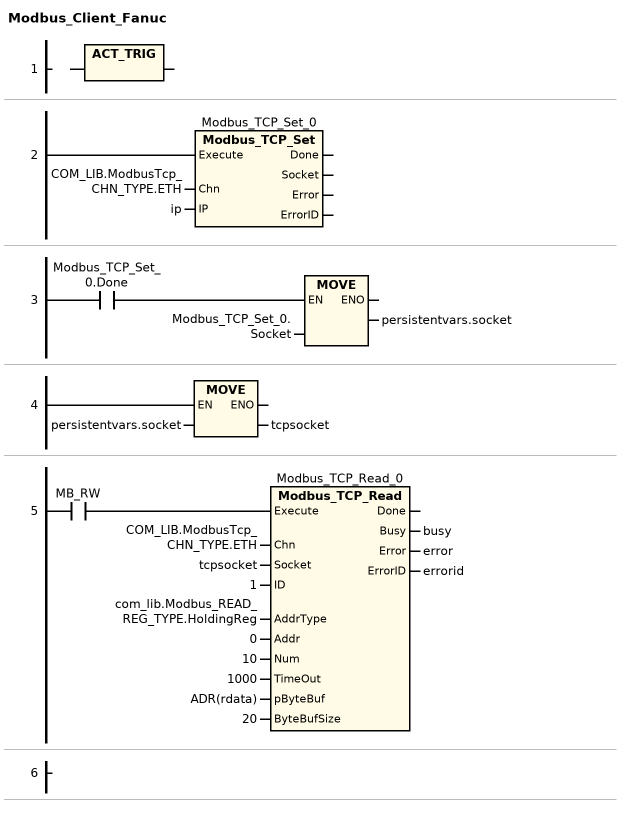
// NETWORK 1
ACT_TRIG();

// NETWORK 2
Modbus_TCP_Set_0(Execute := TRUE, Chn := COM_LIB.ModbusTcp_CHN_TYPE.ETH, IP := ip); // Modbus_TCP_Set

// NETWORK 3
IF Modbus_TCP_Set_0.Done THEN persistentvars.socket := Modbus_TCP_Set_0.Socket; END_IF

// NETWORK 4
tcpsocket := persistentvars.socket;

// NETWORK 5
Modbus_TCP_Read_0(
    Execute := MB_RW,
    Chn := COM_LIB.ModbusTcp_CHN_TYPE.ETH,
    Socket := tcpsocket,
    ID := 1,
    AddrType := com_lib.Modbus_READ_REG_TYPE.HoldingReg,
    Addr := 0,
    Num := 10,
    TimeOut := 1000,
    pByteBuf := ADR(rdata),
    ByteBufSize := 20,
    Busy => busy,
    Error => error,
    ErrorID => errorid); // Modbus_TCP_Read

// NETWORK 6

ACTION ACT_TRIG:


RW(IN:= NOT RW.Q, PT:= T#5MS, Q=> , ET=> );
IF RW.Q=1 THEN 
	MB_RW:=NOT MB_RW;
END_IF
END_ACTION

END_PROGRAM
